DATA_BLOCK "DB242_Program8"   // DB242
{ S7_Optimized_Access := 'FALSE' }
AUTHOR : Robopac
VERSION : 0.0
// stored: AutoNumber false, IsOnlyStoredInLoadMemory false, IsWriteProtectedInAS false
   VAR RETAIN
      Program8 { S7_SetPoint := 'True'} : "DatiProgramma";
   END_VAR
BEGIN
   Program8.Wrapping := TRUE;
   Program8.TopLenght := 500;
   Program8.TopRelease := 0;
   Program8.TopDown := 0;
   Program8.Top := 4;
   Program8.PressurePTime := 0;
   Program8.LifterTime := 0;
   Program8.RevOverContrast := 1;
   Program8.RopeEndCycle := 16#02;
   Program8.Spare4 := 16#01;
   Program8.RopeTime := 1500;
   Program8.RevOverClamp := 1;
   Program8.FilmForceFinalRev := 10;
   Program8.FilmPrestretchFinalRev := 100;
   Program8.ArmSpeed := 100;
   Program8.CarriageDown4Top := 500;
   Program8.TopDownTime := 1500;
   Program8.LapsUnderTop := 0;
   Program8.Spare6 := 0;
   Program8.Spare7 := 0;
   Program8.Spare8 := 0;
   Program8.Spare9 := 0;
   Program8.Spare10 := 0;
   Program8.Spare11 := 0;
   Program8.Spare12 := 0;
   Program8.Overlap0_1 := 0;
   Program8.Height1 := 130;
   Program8.Landmark1 := FALSE;
   Program8.Lifter1 := FALSE;
   Program8.SpareBit1H1 := FALSE;
   Program8.Airblower1 := TRUE;
   Program8.NextStep1 := TRUE;
   Program8.PressureP1 := TRUE;
   Program8.SpareByte2H1 := 16#00;
   Program8.Revolution1 := 1;
   Program8.RopeUnit1_1 := 16#01;
   Program8.RopeUnit1_2 := 16#01;
   Program8.FilmForce1 := 5;
   Program8.FilmPrestretch1 := 200;
   Program8.Spare3H1 := 0;
   Program8.Spare49 := 0;
   Program8.Spare50 := 0;
   Program8.Spare51 := 0;
   Program8.Spare52 := 0;
   Program8.Spare53 := 0;
   Program8.Overlap1_2 := 0;
   Program8.Height2 := 50;
   Program8.Landmark2 := FALSE;
   Program8.Lifter2 := FALSE;
   Program8.SpareBit1H2 := FALSE;
   Program8.Airblower2 := TRUE;
   Program8.NextStep2 := TRUE;
   Program8.PressureP2 := TRUE;
   Program8.SpareByte2H2 := 16#00;
   Program8.Revolution2 := 1;
   Program8.RopeUnit2_1 := 16#01;
   Program8.RopeUnit2_2 := 16#01;
   Program8.FilmForce2 := 20;
   Program8.FilmPrestretch2 := 200;
   Program8.Spare3H2 := 0;
   Program8.Spare54 := 0;
   Program8.Spare55 := 0;
   Program8.Spare56 := 0;
   Program8.Spare57 := 0;
   Program8.Spare58 := 0;
   Program8.Overlap2_3 := 100;
   Program8.Height3 := -50;
   Program8.Landmark3 := TRUE;
   Program8.Lifter3 := FALSE;
   Program8.SpareBit1H3 := FALSE;
   Program8.Airblower3 := TRUE;
   Program8.NextStep3 := TRUE;
   Program8.PressureP3 := TRUE;
   Program8.SpareByte2H3 := 16#00;
   Program8.Revolution3 := 2;
   Program8.RopeUnit3_1 := 16#01;
   Program8.RopeUnit3_2 := 16#01;
   Program8.FilmForce3 := 30;
   Program8.FilmPrestretch3 := 200;
   Program8.Spare3H3 := 0;
   Program8.Spare59 := 0;
   Program8.Spare60 := 0;
   Program8.Spare61 := 380;
   Program8.Spare62 := 2800;
   Program8.Spare63 := 0;
   Program8.Overlap3_4 := 100;
   Program8.Height4 := 100;
   Program8.Landmark4 := FALSE;
   Program8.Lifter4 := FALSE;
   Program8.SpareBit1H4 := FALSE;
   Program8.Airblower4 := TRUE;
   Program8.NextStep4 := TRUE;
   Program8.PressureP4 := TRUE;
   Program8.SpareByte2H4 := 16#00;
   Program8.Revolution4 := 3;
   Program8.RopeUnit4_1 := 16#02;
   Program8.RopeUnit4_2 := 16#02;
   Program8.FilmForce4 := 30;
   Program8.FilmPrestretch4 := 200;
   Program8.Spare3H4 := 0;
   Program8.Spare64 := 0;
   Program8.Spare65 := 0;
   Program8.Spare66 := 0;
   Program8.Spare67 := 0;
   Program8.Spare68 := 0;
   Program8.Overlap4_5 := 0;
   Program8.Height5 := 50;
   Program8.Landmark5 := FALSE;
   Program8.Lifter5 := FALSE;
   Program8.SpareBit1H5 := FALSE;
   Program8.Airblower5 := TRUE;
   Program8.NextStep5 := FALSE;
   Program8.PressureP5 := FALSE;
   Program8.SpareByte2H5 := 16#00;
   Program8.Revolution5 := 1;
   Program8.RopeUnit5_1 := 16#01;
   Program8.RopeUnit5_2 := 16#01;
   Program8.FilmForce5 := 30;
   Program8.FilmPrestretch5 := 200;
   Program8.Spare3H5 := 0;
   Program8.Spare69 := 0;
   Program8.Spare70 := 0;
   Program8.Spare71 := 0;
   Program8.Spare72 := 0;
   Program8.Spare73 := 0;
   Program8.Overlap5_6 := 100;
   Program8.Height6 := 50;
   Program8.Landmark6 := FALSE;
   Program8.Lifter6 := FALSE;
   Program8.SpareBit1H6 := FALSE;
   Program8.Airblower6 := TRUE;
   Program8.NextStep6 := FALSE;
   Program8.PressureP6 := FALSE;
   Program8.SpareByte2H6 := 16#00;
   Program8.Revolution6 := 2;
   Program8.RopeUnit6_1 := 16#02;
   Program8.RopeUnit6_2 := 16#01;
   Program8.FilmForce6 := 20;
   Program8.FilmPrestretch6 := 200;
   Program8.Spare3H6 := 0;
   Program8.Spare74 := 0;
   Program8.Spare75 := 0;
   Program8.Spare76 := 0;
   Program8.Spare77 := 0;
   Program8.Spare78 := 0;
   Program8.Overlap6_7 := 0;
   Program8.Height7 := 0;
   Program8.Landmark7 := FALSE;
   Program8.Lifter7 := FALSE;
   Program8.SpareBit1H7 := FALSE;
   Program8.Airblower7 := FALSE;
   Program8.NextStep7 := TRUE;
   Program8.PressureP7 := FALSE;
   Program8.SpareByte2H7 := 16#00;
   Program8.Revolution7 := 1;
   Program8.RopeUnit7_1 := 16#01;
   Program8.RopeUnit7_2 := 16#01;
   Program8.FilmForce7 := 0;
   Program8.FilmPrestretch7 := 100;
   Program8.Spare3H7 := 0;
   Program8.Spare79 := 0;
   Program8.Spare80 := 0;
   Program8.Spare81 := 0;
   Program8.Spare82 := 0;
   Program8.Spare83 := 0;
   Program8.Overlap7_8 := 0;
   Program8.Height8 := 0;
   Program8.Landmark8 := FALSE;
   Program8.Lifter8 := FALSE;
   Program8.SpareBit1H8 := FALSE;
   Program8.Airblower8 := FALSE;
   Program8.NextStep8 := TRUE;
   Program8.PressureP8 := FALSE;
   Program8.SpareByte2H8 := 16#00;
   Program8.Revolution8 := 1;
   Program8.RopeUnit8_1 := 16#01;
   Program8.RopeUnit8_2 := 16#01;
   Program8.FilmForce8 := 0;
   Program8.FilmPrestretch8 := 100;
   Program8.Spare3H8 := 0;
   Program8.Spare84 := 0;
   Program8.Spare85 := 0;
   Program8.Spare86 := 0;
   Program8.Spare87 := 0;
   Program8.Spare88 := 0;
   Program8.Overlap8_9 := 0;
   Program8.Height9 := 0;
   Program8.Landmark9 := FALSE;
   Program8.Lifter9 := FALSE;
   Program8.SpareBit1H9 := FALSE;
   Program8.Airblower9 := FALSE;
   Program8.NextStep9 := TRUE;
   Program8.PressureP9 := FALSE;
   Program8.SpareByte2H9 := 16#00;
   Program8.Revolution9 := 1;
   Program8.RopeUnit9_1 := 16#01;
   Program8.RopeUnit9_2 := 16#01;
   Program8.FilmForce9 := 0;
   Program8.FilmPrestretch9 := 100;
   Program8.Spare3H9 := 0;
   Program8.Spare89 := 0;
   Program8.Spare90 := 0;
   Program8.Spare91 := 0;
   Program8.Spare92 := 0;
   Program8.Spare93 := 0;
   Program8.Overlap9_10 := 0;
   Program8.Height10 := 0;
   Program8.Landmark10 := FALSE;
   Program8.Lifter10 := FALSE;
   Program8.SpareBit1H10 := FALSE;
   Program8.Airblower10 := FALSE;
   Program8.NextStep10 := FALSE;
   Program8.PressureP10 := FALSE;
   Program8.SpareByte2H10 := 16#00;
   Program8.Revolution10 := 1;
   Program8.RopeUnit10_1 := 16#01;
   Program8.RopeUnit10_2 := 16#01;
   Program8.FilmForce10 := 0;
   Program8.FilmPrestretch10 := 100;
   Program8.Spare3H10 := 0;
   Program8.Spare94 := 0;
   Program8.Spare95 := 0;
   Program8.Spare96 := 0;
   Program8.Spare97 := 0;
   Program8.Spare98 := 0;
   Program8.Overlap10_11 := 0;
   Program8.Height11 := 0;
   Program8.Landmark11 := FALSE;
   Program8.Lifter11 := FALSE;
   Program8.SpareBit1H11 := FALSE;
   Program8.Airblower11 := FALSE;
   Program8.NextStep11 := TRUE;
   Program8.PressureP11 := FALSE;
   Program8.SpareByte2H11 := 16#00;
   Program8.Revolution11 := 1;
   Program8.RopeUnit11_1 := 16#01;
   Program8.RopeUnit11_2 := 16#01;
   Program8.FilmForce11 := 0;
   Program8.FilmPrestretch11 := 100;
   Program8.Spare3H11 := 0;
   Program8.Spare99 := 0;
   Program8.Spare100 := 0;
   Program8.Spare101 := 0;
   Program8.Spare102 := 0;
   Program8.Spare103 := 0;
   Program8.Overlap11_12 := 0;
   Program8.Height12 := 0;
   Program8.Landmark12 := FALSE;
   Program8.Lifter12 := FALSE;
   Program8.SpareBit1H12 := FALSE;
   Program8.Airblower12 := FALSE;
   Program8.NextStep12 := FALSE;
   Program8.PressureP12 := FALSE;
   Program8.SpareByte2H12 := 16#00;
   Program8.Revolution12 := 1;
   Program8.RopeUnit12_1 := 16#01;
   Program8.RopeUnit12_2 := 16#01;
   Program8.FilmForce12 := 0;
   Program8.FilmPrestretch12 := 100;
   Program8.Spare3H12 := 0;
   Program8.Spare104 := 0;
   Program8.Spare105 := 0;
   Program8.Spare106 := 0;
   Program8.Spare107 := 0;
   Program8.Spare108 := 0;
END_DATA_BLOCK

DATA_BLOCK "DB244_Program6"   // DB244
{ S7_Optimized_Access := 'FALSE' }
AUTHOR : Robopac
VERSION : 0.0
// stored: AutoNumber false, IsOnlyStoredInLoadMemory false, IsWriteProtectedInAS false
   VAR RETAIN
      Program6 { S7_SetPoint := 'True'} : "DatiProgramma";
   END_VAR
BEGIN
   Program6.Wrapping := TRUE;
   Program6.TopLenght := 500;
   Program6.TopRelease := 0;
   Program6.TopDown := 0;
   Program6.Top := 4;
   Program6.PressurePTime := 0;
   Program6.LifterTime := 0;
   Program6.RevOverContrast := 1;
   Program6.RopeEndCycle := 16#02;
   Program6.Spare4 := 16#01;
   Program6.RopeTime := 1500;
   Program6.RevOverClamp := 1;
   Program6.FilmForceFinalRev := 10;
   Program6.FilmPrestretchFinalRev := 100;
   Program6.ArmSpeed := 100;
   Program6.CarriageDown4Top := 500;
   Program6.TopDownTime := 1500;
   Program6.LapsUnderTop := 0;
   Program6.Spare6 := 0;
   Program6.Spare7 := 0;
   Program6.Spare8 := 0;
   Program6.Spare9 := 0;
   Program6.Spare10 := 0;
   Program6.Spare11 := 0;
   Program6.Spare12 := 0;
   Program6.Overlap0_1 := 0;
   Program6.Height1 := 130;
   Program6.Landmark1 := FALSE;
   Program6.Lifter1 := FALSE;
   Program6.SpareBit1H1 := FALSE;
   Program6.Airblower1 := TRUE;
   Program6.NextStep1 := TRUE;
   Program6.PressureP1 := TRUE;
   Program6.SpareByte2H1 := 16#00;
   Program6.Revolution1 := 1;
   Program6.RopeUnit1_1 := 16#01;
   Program6.RopeUnit1_2 := 16#01;
   Program6.FilmForce1 := 5;
   Program6.FilmPrestretch1 := 200;
   Program6.Spare3H1 := 0;
   Program6.Spare49 := 0;
   Program6.Spare50 := 0;
   Program6.Spare51 := 0;
   Program6.Spare52 := 0;
   Program6.Spare53 := 0;
   Program6.Overlap1_2 := 0;
   Program6.Height2 := 50;
   Program6.Landmark2 := FALSE;
   Program6.Lifter2 := FALSE;
   Program6.SpareBit1H2 := FALSE;
   Program6.Airblower2 := TRUE;
   Program6.NextStep2 := TRUE;
   Program6.PressureP2 := TRUE;
   Program6.SpareByte2H2 := 16#00;
   Program6.Revolution2 := 1;
   Program6.RopeUnit2_1 := 16#01;
   Program6.RopeUnit2_2 := 16#01;
   Program6.FilmForce2 := 20;
   Program6.FilmPrestretch2 := 200;
   Program6.Spare3H2 := 0;
   Program6.Spare54 := 0;
   Program6.Spare55 := 0;
   Program6.Spare56 := 0;
   Program6.Spare57 := 0;
   Program6.Spare58 := 0;
   Program6.Overlap2_3 := 100;
   Program6.Height3 := -50;
   Program6.Landmark3 := TRUE;
   Program6.Lifter3 := FALSE;
   Program6.SpareBit1H3 := FALSE;
   Program6.Airblower3 := TRUE;
   Program6.NextStep3 := TRUE;
   Program6.PressureP3 := TRUE;
   Program6.SpareByte2H3 := 16#00;
   Program6.Revolution3 := 2;
   Program6.RopeUnit3_1 := 16#01;
   Program6.RopeUnit3_2 := 16#01;
   Program6.FilmForce3 := 30;
   Program6.FilmPrestretch3 := 200;
   Program6.Spare3H3 := 0;
   Program6.Spare59 := 0;
   Program6.Spare60 := 0;
   Program6.Spare61 := 380;
   Program6.Spare62 := 2800;
   Program6.Spare63 := 0;
   Program6.Overlap3_4 := 100;
   Program6.Height4 := 100;
   Program6.Landmark4 := FALSE;
   Program6.Lifter4 := FALSE;
   Program6.SpareBit1H4 := FALSE;
   Program6.Airblower4 := TRUE;
   Program6.NextStep4 := TRUE;
   Program6.PressureP4 := TRUE;
   Program6.SpareByte2H4 := 16#00;
   Program6.Revolution4 := 3;
   Program6.RopeUnit4_1 := 16#02;
   Program6.RopeUnit4_2 := 16#02;
   Program6.FilmForce4 := 30;
   Program6.FilmPrestretch4 := 200;
   Program6.Spare3H4 := 0;
   Program6.Spare64 := 0;
   Program6.Spare65 := 0;
   Program6.Spare66 := 0;
   Program6.Spare67 := 0;
   Program6.Spare68 := 0;
   Program6.Overlap4_5 := 0;
   Program6.Height5 := 50;
   Program6.Landmark5 := FALSE;
   Program6.Lifter5 := FALSE;
   Program6.SpareBit1H5 := FALSE;
   Program6.Airblower5 := TRUE;
   Program6.NextStep5 := FALSE;
   Program6.PressureP5 := FALSE;
   Program6.SpareByte2H5 := 16#00;
   Program6.Revolution5 := 1;
   Program6.RopeUnit5_1 := 16#01;
   Program6.RopeUnit5_2 := 16#01;
   Program6.FilmForce5 := 30;
   Program6.FilmPrestretch5 := 200;
   Program6.Spare3H5 := 0;
   Program6.Spare69 := 0;
   Program6.Spare70 := 0;
   Program6.Spare71 := 0;
   Program6.Spare72 := 0;
   Program6.Spare73 := 0;
   Program6.Overlap5_6 := 100;
   Program6.Height6 := 50;
   Program6.Landmark6 := FALSE;
   Program6.Lifter6 := FALSE;
   Program6.SpareBit1H6 := FALSE;
   Program6.Airblower6 := TRUE;
   Program6.NextStep6 := FALSE;
   Program6.PressureP6 := FALSE;
   Program6.SpareByte2H6 := 16#00;
   Program6.Revolution6 := 2;
   Program6.RopeUnit6_1 := 16#02;
   Program6.RopeUnit6_2 := 16#01;
   Program6.FilmForce6 := 20;
   Program6.FilmPrestretch6 := 200;
   Program6.Spare3H6 := 0;
   Program6.Spare74 := 0;
   Program6.Spare75 := 0;
   Program6.Spare76 := 0;
   Program6.Spare77 := 0;
   Program6.Spare78 := 0;
   Program6.Overlap6_7 := 0;
   Program6.Height7 := 0;
   Program6.Landmark7 := FALSE;
   Program6.Lifter7 := FALSE;
   Program6.SpareBit1H7 := FALSE;
   Program6.Airblower7 := FALSE;
   Program6.NextStep7 := TRUE;
   Program6.PressureP7 := FALSE;
   Program6.SpareByte2H7 := 16#00;
   Program6.Revolution7 := 1;
   Program6.RopeUnit7_1 := 16#01;
   Program6.RopeUnit7_2 := 16#01;
   Program6.FilmForce7 := 0;
   Program6.FilmPrestretch7 := 100;
   Program6.Spare3H7 := 0;
   Program6.Spare79 := 0;
   Program6.Spare80 := 0;
   Program6.Spare81 := 0;
   Program6.Spare82 := 0;
   Program6.Spare83 := 0;
   Program6.Overlap7_8 := 0;
   Program6.Height8 := 0;
   Program6.Landmark8 := FALSE;
   Program6.Lifter8 := FALSE;
   Program6.SpareBit1H8 := FALSE;
   Program6.Airblower8 := FALSE;
   Program6.NextStep8 := TRUE;
   Program6.PressureP8 := FALSE;
   Program6.SpareByte2H8 := 16#00;
   Program6.Revolution8 := 1;
   Program6.RopeUnit8_1 := 16#01;
   Program6.RopeUnit8_2 := 16#01;
   Program6.FilmForce8 := 0;
   Program6.FilmPrestretch8 := 100;
   Program6.Spare3H8 := 0;
   Program6.Spare84 := 0;
   Program6.Spare85 := 0;
   Program6.Spare86 := 0;
   Program6.Spare87 := 0;
   Program6.Spare88 := 0;
   Program6.Overlap8_9 := 0;
   Program6.Height9 := 0;
   Program6.Landmark9 := FALSE;
   Program6.Lifter9 := FALSE;
   Program6.SpareBit1H9 := FALSE;
   Program6.Airblower9 := FALSE;
   Program6.NextStep9 := TRUE;
   Program6.PressureP9 := FALSE;
   Program6.SpareByte2H9 := 16#00;
   Program6.Revolution9 := 1;
   Program6.RopeUnit9_1 := 16#01;
   Program6.RopeUnit9_2 := 16#01;
   Program6.FilmForce9 := 0;
   Program6.FilmPrestretch9 := 100;
   Program6.Spare3H9 := 0;
   Program6.Spare89 := 0;
   Program6.Spare90 := 0;
   Program6.Spare91 := 0;
   Program6.Spare92 := 0;
   Program6.Spare93 := 0;
   Program6.Overlap9_10 := 0;
   Program6.Height10 := 0;
   Program6.Landmark10 := FALSE;
   Program6.Lifter10 := FALSE;
   Program6.SpareBit1H10 := FALSE;
   Program6.Airblower10 := FALSE;
   Program6.NextStep10 := FALSE;
   Program6.PressureP10 := FALSE;
   Program6.SpareByte2H10 := 16#00;
   Program6.Revolution10 := 1;
   Program6.RopeUnit10_1 := 16#01;
   Program6.RopeUnit10_2 := 16#01;
   Program6.FilmForce10 := 0;
   Program6.FilmPrestretch10 := 100;
   Program6.Spare3H10 := 0;
   Program6.Spare94 := 0;
   Program6.Spare95 := 0;
   Program6.Spare96 := 0;
   Program6.Spare97 := 0;
   Program6.Spare98 := 0;
   Program6.Overlap10_11 := 0;
   Program6.Height11 := 0;
   Program6.Landmark11 := FALSE;
   Program6.Lifter11 := FALSE;
   Program6.SpareBit1H11 := FALSE;
   Program6.Airblower11 := FALSE;
   Program6.NextStep11 := TRUE;
   Program6.PressureP11 := FALSE;
   Program6.SpareByte2H11 := 16#00;
   Program6.Revolution11 := 1;
   Program6.RopeUnit11_1 := 16#01;
   Program6.RopeUnit11_2 := 16#01;
   Program6.FilmForce11 := 0;
   Program6.FilmPrestretch11 := 100;
   Program6.Spare3H11 := 0;
   Program6.Spare99 := 0;
   Program6.Spare100 := 0;
   Program6.Spare101 := 0;
   Program6.Spare102 := 0;
   Program6.Spare103 := 0;
   Program6.Overlap11_12 := 0;
   Program6.Height12 := 0;
   Program6.Landmark12 := FALSE;
   Program6.Lifter12 := FALSE;
   Program6.SpareBit1H12 := FALSE;
   Program6.Airblower12 := FALSE;
   Program6.NextStep12 := FALSE;
   Program6.PressureP12 := FALSE;
   Program6.SpareByte2H12 := 16#00;
   Program6.Revolution12 := 1;
   Program6.RopeUnit12_1 := 16#01;
   Program6.RopeUnit12_2 := 16#01;
   Program6.FilmForce12 := 0;
   Program6.FilmPrestretch12 := 100;
   Program6.Spare3H12 := 0;
   Program6.Spare104 := 0;
   Program6.Spare105 := 0;
   Program6.Spare106 := 0;
   Program6.Spare107 := 0;
   Program6.Spare108 := 0;
END_DATA_BLOCK

DATA_BLOCK "DB245_Program5"   // DB245
{ S7_Optimized_Access := 'FALSE' }
AUTHOR : Robopac
VERSION : 0.0
// stored: AutoNumber false, IsOnlyStoredInLoadMemory false, IsWriteProtectedInAS false
   VAR RETAIN
      Program5 { S7_SetPoint := 'True'} : "DatiProgramma";
   END_VAR
BEGIN
   Program5.Wrapping := TRUE;
   Program5.TopLenght := 500;
   Program5.TopRelease := 0;
   Program5.TopDown := 0;
   Program5.Top := 4;
   Program5.PressurePTime := 0;
   Program5.LifterTime := 0;
   Program5.RevOverContrast := 1;
   Program5.RopeEndCycle := 16#02;
   Program5.Spare4 := 16#01;
   Program5.RopeTime := 1500;
   Program5.RevOverClamp := 1;
   Program5.FilmForceFinalRev := 10;
   Program5.FilmPrestretchFinalRev := 100;
   Program5.ArmSpeed := 100;
   Program5.CarriageDown4Top := 500;
   Program5.TopDownTime := 1500;
   Program5.LapsUnderTop := 0;
   Program5.Spare6 := 0;
   Program5.Spare7 := 0;
   Program5.Spare8 := 0;
   Program5.Spare9 := 0;
   Program5.Spare10 := 0;
   Program5.Spare11 := 0;
   Program5.Spare12 := 0;
   Program5.Overlap0_1 := 0;
   Program5.Height1 := 130;
   Program5.Landmark1 := FALSE;
   Program5.Lifter1 := FALSE;
   Program5.SpareBit1H1 := FALSE;
   Program5.Airblower1 := TRUE;
   Program5.NextStep1 := TRUE;
   Program5.PressureP1 := TRUE;
   Program5.SpareByte2H1 := 16#00;
   Program5.Revolution1 := 1;
   Program5.RopeUnit1_1 := 16#01;
   Program5.RopeUnit1_2 := 16#01;
   Program5.FilmForce1 := 5;
   Program5.FilmPrestretch1 := 200;
   Program5.Spare3H1 := 0;
   Program5.Spare49 := 0;
   Program5.Spare50 := 0;
   Program5.Spare51 := 0;
   Program5.Spare52 := 0;
   Program5.Spare53 := 0;
   Program5.Overlap1_2 := 0;
   Program5.Height2 := 50;
   Program5.Landmark2 := FALSE;
   Program5.Lifter2 := FALSE;
   Program5.SpareBit1H2 := FALSE;
   Program5.Airblower2 := TRUE;
   Program5.NextStep2 := TRUE;
   Program5.PressureP2 := TRUE;
   Program5.SpareByte2H2 := 16#00;
   Program5.Revolution2 := 1;
   Program5.RopeUnit2_1 := 16#01;
   Program5.RopeUnit2_2 := 16#01;
   Program5.FilmForce2 := 20;
   Program5.FilmPrestretch2 := 200;
   Program5.Spare3H2 := 0;
   Program5.Spare54 := 0;
   Program5.Spare55 := 0;
   Program5.Spare56 := 0;
   Program5.Spare57 := 0;
   Program5.Spare58 := 0;
   Program5.Overlap2_3 := 100;
   Program5.Height3 := -50;
   Program5.Landmark3 := TRUE;
   Program5.Lifter3 := FALSE;
   Program5.SpareBit1H3 := FALSE;
   Program5.Airblower3 := TRUE;
   Program5.NextStep3 := TRUE;
   Program5.PressureP3 := TRUE;
   Program5.SpareByte2H3 := 16#00;
   Program5.Revolution3 := 2;
   Program5.RopeUnit3_1 := 16#01;
   Program5.RopeUnit3_2 := 16#01;
   Program5.FilmForce3 := 30;
   Program5.FilmPrestretch3 := 200;
   Program5.Spare3H3 := 0;
   Program5.Spare59 := 0;
   Program5.Spare60 := 0;
   Program5.Spare61 := 380;
   Program5.Spare62 := 2800;
   Program5.Spare63 := 0;
   Program5.Overlap3_4 := 100;
   Program5.Height4 := 100;
   Program5.Landmark4 := FALSE;
   Program5.Lifter4 := FALSE;
   Program5.SpareBit1H4 := FALSE;
   Program5.Airblower4 := TRUE;
   Program5.NextStep4 := TRUE;
   Program5.PressureP4 := TRUE;
   Program5.SpareByte2H4 := 16#00;
   Program5.Revolution4 := 3;
   Program5.RopeUnit4_1 := 16#02;
   Program5.RopeUnit4_2 := 16#02;
   Program5.FilmForce4 := 30;
   Program5.FilmPrestretch4 := 200;
   Program5.Spare3H4 := 0;
   Program5.Spare64 := 0;
   Program5.Spare65 := 0;
   Program5.Spare66 := 0;
   Program5.Spare67 := 0;
   Program5.Spare68 := 0;
   Program5.Overlap4_5 := 0;
   Program5.Height5 := 50;
   Program5.Landmark5 := FALSE;
   Program5.Lifter5 := FALSE;
   Program5.SpareBit1H5 := FALSE;
   Program5.Airblower5 := TRUE;
   Program5.NextStep5 := FALSE;
   Program5.PressureP5 := FALSE;
   Program5.SpareByte2H5 := 16#00;
   Program5.Revolution5 := 1;
   Program5.RopeUnit5_1 := 16#01;
   Program5.RopeUnit5_2 := 16#01;
   Program5.FilmForce5 := 30;
   Program5.FilmPrestretch5 := 200;
   Program5.Spare3H5 := 0;
   Program5.Spare69 := 0;
   Program5.Spare70 := 0;
   Program5.Spare71 := 0;
   Program5.Spare72 := 0;
   Program5.Spare73 := 0;
   Program5.Overlap5_6 := 100;
   Program5.Height6 := 50;
   Program5.Landmark6 := FALSE;
   Program5.Lifter6 := FALSE;
   Program5.SpareBit1H6 := FALSE;
   Program5.Airblower6 := TRUE;
   Program5.NextStep6 := FALSE;
   Program5.PressureP6 := FALSE;
   Program5.SpareByte2H6 := 16#00;
   Program5.Revolution6 := 2;
   Program5.RopeUnit6_1 := 16#02;
   Program5.RopeUnit6_2 := 16#01;
   Program5.FilmForce6 := 20;
   Program5.FilmPrestretch6 := 200;
   Program5.Spare3H6 := 0;
   Program5.Spare74 := 0;
   Program5.Spare75 := 0;
   Program5.Spare76 := 0;
   Program5.Spare77 := 0;
   Program5.Spare78 := 0;
   Program5.Overlap6_7 := 0;
   Program5.Height7 := 0;
   Program5.Landmark7 := FALSE;
   Program5.Lifter7 := FALSE;
   Program5.SpareBit1H7 := FALSE;
   Program5.Airblower7 := FALSE;
   Program5.NextStep7 := TRUE;
   Program5.PressureP7 := FALSE;
   Program5.SpareByte2H7 := 16#00;
   Program5.Revolution7 := 1;
   Program5.RopeUnit7_1 := 16#01;
   Program5.RopeUnit7_2 := 16#01;
   Program5.FilmForce7 := 0;
   Program5.FilmPrestretch7 := 100;
   Program5.Spare3H7 := 0;
   Program5.Spare79 := 0;
   Program5.Spare80 := 0;
   Program5.Spare81 := 0;
   Program5.Spare82 := 0;
   Program5.Spare83 := 0;
   Program5.Overlap7_8 := 0;
   Program5.Height8 := 0;
   Program5.Landmark8 := FALSE;
   Program5.Lifter8 := FALSE;
   Program5.SpareBit1H8 := FALSE;
   Program5.Airblower8 := FALSE;
   Program5.NextStep8 := TRUE;
   Program5.PressureP8 := FALSE;
   Program5.SpareByte2H8 := 16#00;
   Program5.Revolution8 := 1;
   Program5.RopeUnit8_1 := 16#01;
   Program5.RopeUnit8_2 := 16#01;
   Program5.FilmForce8 := 0;
   Program5.FilmPrestretch8 := 100;
   Program5.Spare3H8 := 0;
   Program5.Spare84 := 0;
   Program5.Spare85 := 0;
   Program5.Spare86 := 0;
   Program5.Spare87 := 0;
   Program5.Spare88 := 0;
   Program5.Overlap8_9 := 0;
   Program5.Height9 := 0;
   Program5.Landmark9 := FALSE;
   Program5.Lifter9 := FALSE;
   Program5.SpareBit1H9 := FALSE;
   Program5.Airblower9 := FALSE;
   Program5.NextStep9 := TRUE;
   Program5.PressureP9 := FALSE;
   Program5.SpareByte2H9 := 16#00;
   Program5.Revolution9 := 1;
   Program5.RopeUnit9_1 := 16#01;
   Program5.RopeUnit9_2 := 16#01;
   Program5.FilmForce9 := 0;
   Program5.FilmPrestretch9 := 100;
   Program5.Spare3H9 := 0;
   Program5.Spare89 := 0;
   Program5.Spare90 := 0;
   Program5.Spare91 := 0;
   Program5.Spare92 := 0;
   Program5.Spare93 := 0;
   Program5.Overlap9_10 := 0;
   Program5.Height10 := 0;
   Program5.Landmark10 := FALSE;
   Program5.Lifter10 := FALSE;
   Program5.SpareBit1H10 := FALSE;
   Program5.Airblower10 := FALSE;
   Program5.NextStep10 := FALSE;
   Program5.PressureP10 := FALSE;
   Program5.SpareByte2H10 := 16#00;
   Program5.Revolution10 := 1;
   Program5.RopeUnit10_1 := 16#01;
   Program5.RopeUnit10_2 := 16#01;
   Program5.FilmForce10 := 0;
   Program5.FilmPrestretch10 := 100;
   Program5.Spare3H10 := 0;
   Program5.Spare94 := 0;
   Program5.Spare95 := 0;
   Program5.Spare96 := 0;
   Program5.Spare97 := 0;
   Program5.Spare98 := 0;
   Program5.Overlap10_11 := 0;
   Program5.Height11 := 0;
   Program5.Landmark11 := FALSE;
   Program5.Lifter11 := FALSE;
   Program5.SpareBit1H11 := FALSE;
   Program5.Airblower11 := FALSE;
   Program5.NextStep11 := TRUE;
   Program5.PressureP11 := FALSE;
   Program5.SpareByte2H11 := 16#00;
   Program5.Revolution11 := 1;
   Program5.RopeUnit11_1 := 16#01;
   Program5.RopeUnit11_2 := 16#01;
   Program5.FilmForce11 := 0;
   Program5.FilmPrestretch11 := 100;
   Program5.Spare3H11 := 0;
   Program5.Spare99 := 0;
   Program5.Spare100 := 0;
   Program5.Spare101 := 0;
   Program5.Spare102 := 0;
   Program5.Spare103 := 0;
   Program5.Overlap11_12 := 0;
   Program5.Height12 := 0;
   Program5.Landmark12 := FALSE;
   Program5.Lifter12 := FALSE;
   Program5.SpareBit1H12 := FALSE;
   Program5.Airblower12 := FALSE;
   Program5.NextStep12 := FALSE;
   Program5.PressureP12 := FALSE;
   Program5.SpareByte2H12 := 16#00;
   Program5.Revolution12 := 1;
   Program5.RopeUnit12_1 := 16#01;
   Program5.RopeUnit12_2 := 16#01;
   Program5.FilmForce12 := 0;
   Program5.FilmPrestretch12 := 100;
   Program5.Spare3H12 := 0;
   Program5.Spare104 := 0;
   Program5.Spare105 := 0;
   Program5.Spare106 := 0;
   Program5.Spare107 := 0;
   Program5.Spare108 := 0;
END_DATA_BLOCK

DATA_BLOCK "DB247_Program3"   // DB247
{ S7_Optimized_Access := 'FALSE' }
AUTHOR : Robopac
VERSION : 0.0
// stored: AutoNumber false, IsOnlyStoredInLoadMemory false, IsWriteProtectedInAS false
   VAR RETAIN
      Program3 { S7_SetPoint := 'True'} : "DatiProgramma";
   END_VAR
BEGIN
   Program3.Wrapping := TRUE;
   Program3.TopLenght := 500;
   Program3.TopRelease := 0;
   Program3.TopDown := 0;
   Program3.Top := 4;
   Program3.PressurePTime := 0;
   Program3.LifterTime := 0;
   Program3.RevOverContrast := 1;
   Program3.RopeEndCycle := 16#01;
   Program3.Spare4 := 16#01;
   Program3.RopeTime := 1500;
   Program3.RevOverClamp := 1;
   Program3.FilmForceFinalRev := 20;
   Program3.FilmPrestretchFinalRev := 100;
   Program3.ArmSpeed := 90;
   Program3.CarriageDown4Top := 500;
   Program3.TopDownTime := 1500;
   Program3.LapsUnderTop := 0;
   Program3.Spare6 := 0;
   Program3.Spare7 := 0;
   Program3.Spare8 := 0;
   Program3.Spare9 := 0;
   Program3.Spare10 := 0;
   Program3.Spare11 := 0;
   Program3.Spare12 := 0;
   Program3.Overlap0_1 := 0;
   Program3.Height1 := 120;
   Program3.Landmark1 := FALSE;
   Program3.Lifter1 := FALSE;
   Program3.SpareBit1H1 := FALSE;
   Program3.Airblower1 := TRUE;
   Program3.NextStep1 := TRUE;
   Program3.PressureP1 := TRUE;
   Program3.SpareByte2H1 := 16#00;
   Program3.Revolution1 := 1;
   Program3.RopeUnit1_1 := 16#01;
   Program3.RopeUnit1_2 := 16#01;
   Program3.FilmForce1 := 5;
   Program3.FilmPrestretch1 := 200;
   Program3.Spare3H1 := 0;
   Program3.Spare49 := 0;
   Program3.Spare50 := 0;
   Program3.Spare51 := 0;
   Program3.Spare52 := 0;
   Program3.Spare53 := 0;
   Program3.Overlap1_2 := 0;
   Program3.Height2 := 60;
   Program3.Landmark2 := FALSE;
   Program3.Lifter2 := FALSE;
   Program3.SpareBit1H2 := FALSE;
   Program3.Airblower2 := TRUE;
   Program3.NextStep2 := TRUE;
   Program3.PressureP2 := TRUE;
   Program3.SpareByte2H2 := 16#00;
   Program3.Revolution2 := 3;
   Program3.RopeUnit2_1 := 16#01;
   Program3.RopeUnit2_2 := 16#01;
   Program3.FilmForce2 := 10;
   Program3.FilmPrestretch2 := 200;
   Program3.Spare3H2 := 0;
   Program3.Spare54 := 0;
   Program3.Spare55 := 0;
   Program3.Spare56 := 0;
   Program3.Spare57 := 0;
   Program3.Spare58 := 0;
   Program3.Overlap2_3 := 100;
   Program3.Height3 := 120;
   Program3.Landmark3 := FALSE;
   Program3.Lifter3 := FALSE;
   Program3.SpareBit1H3 := FALSE;
   Program3.Airblower3 := TRUE;
   Program3.NextStep3 := TRUE;
   Program3.PressureP3 := TRUE;
   Program3.SpareByte2H3 := 16#00;
   Program3.Revolution3 := 2;
   Program3.RopeUnit3_1 := 16#01;
   Program3.RopeUnit3_2 := 16#01;
   Program3.FilmForce3 := 5;
   Program3.FilmPrestretch3 := 200;
   Program3.Spare3H3 := 0;
   Program3.Spare59 := 0;
   Program3.Spare60 := 0;
   Program3.Spare61 := 380;
   Program3.Spare62 := 2800;
   Program3.Spare63 := 0;
   Program3.Overlap3_4 := 200;
   Program3.Height4 := 120;
   Program3.Landmark4 := FALSE;
   Program3.Lifter4 := FALSE;
   Program3.SpareBit1H4 := FALSE;
   Program3.Airblower4 := TRUE;
   Program3.NextStep4 := TRUE;
   Program3.PressureP4 := TRUE;
   Program3.SpareByte2H4 := 16#00;
   Program3.Revolution4 := 1;
   Program3.RopeUnit4_1 := 16#01;
   Program3.RopeUnit4_2 := 16#01;
   Program3.FilmForce4 := 20;
   Program3.FilmPrestretch4 := 200;
   Program3.Spare3H4 := 0;
   Program3.Spare64 := 0;
   Program3.Spare65 := 0;
   Program3.Spare66 := 0;
   Program3.Spare67 := 0;
   Program3.Spare68 := 0;
   Program3.Overlap4_5 := 200;
   Program3.Height5 := -150;
   Program3.Landmark5 := TRUE;
   Program3.Lifter5 := FALSE;
   Program3.SpareBit1H5 := FALSE;
   Program3.Airblower5 := FALSE;
   Program3.NextStep5 := TRUE;
   Program3.PressureP5 := FALSE;
   Program3.SpareByte2H5 := 16#00;
   Program3.Revolution5 := 1;
   Program3.RopeUnit5_1 := 16#01;
   Program3.RopeUnit5_2 := 16#01;
   Program3.FilmForce5 := 20;
   Program3.FilmPrestretch5 := 200;
   Program3.Spare3H5 := 0;
   Program3.Spare69 := 0;
   Program3.Spare70 := 0;
   Program3.Spare71 := 0;
   Program3.Spare72 := 0;
   Program3.Spare73 := 0;
   Program3.Overlap5_6 := 100;
   Program3.Height6 := 0;
   Program3.Landmark6 := FALSE;
   Program3.Lifter6 := FALSE;
   Program3.SpareBit1H6 := FALSE;
   Program3.Airblower6 := FALSE;
   Program3.NextStep6 := FALSE;
   Program3.PressureP6 := FALSE;
   Program3.SpareByte2H6 := 16#00;
   Program3.Revolution6 := 1;
   Program3.RopeUnit6_1 := 16#01;
   Program3.RopeUnit6_2 := 16#01;
   Program3.FilmForce6 := 30;
   Program3.FilmPrestretch6 := 200;
   Program3.Spare3H6 := 0;
   Program3.Spare74 := 0;
   Program3.Spare75 := 0;
   Program3.Spare76 := 0;
   Program3.Spare77 := 0;
   Program3.Spare78 := 0;
   Program3.Overlap6_7 := 0;
   Program3.Height7 := 0;
   Program3.Landmark7 := FALSE;
   Program3.Lifter7 := FALSE;
   Program3.SpareBit1H7 := FALSE;
   Program3.Airblower7 := FALSE;
   Program3.NextStep7 := TRUE;
   Program3.PressureP7 := FALSE;
   Program3.SpareByte2H7 := 16#00;
   Program3.Revolution7 := 1;
   Program3.RopeUnit7_1 := 16#01;
   Program3.RopeUnit7_2 := 16#01;
   Program3.FilmForce7 := 0;
   Program3.FilmPrestretch7 := 100;
   Program3.Spare3H7 := 0;
   Program3.Spare79 := 0;
   Program3.Spare80 := 0;
   Program3.Spare81 := 0;
   Program3.Spare82 := 0;
   Program3.Spare83 := 0;
   Program3.Overlap7_8 := 0;
   Program3.Height8 := 0;
   Program3.Landmark8 := FALSE;
   Program3.Lifter8 := FALSE;
   Program3.SpareBit1H8 := FALSE;
   Program3.Airblower8 := FALSE;
   Program3.NextStep8 := TRUE;
   Program3.PressureP8 := FALSE;
   Program3.SpareByte2H8 := 16#00;
   Program3.Revolution8 := 1;
   Program3.RopeUnit8_1 := 16#01;
   Program3.RopeUnit8_2 := 16#01;
   Program3.FilmForce8 := 0;
   Program3.FilmPrestretch8 := 100;
   Program3.Spare3H8 := 0;
   Program3.Spare84 := 0;
   Program3.Spare85 := 0;
   Program3.Spare86 := 0;
   Program3.Spare87 := 0;
   Program3.Spare88 := 0;
   Program3.Overlap8_9 := 0;
   Program3.Height9 := 0;
   Program3.Landmark9 := FALSE;
   Program3.Lifter9 := FALSE;
   Program3.SpareBit1H9 := FALSE;
   Program3.Airblower9 := FALSE;
   Program3.NextStep9 := TRUE;
   Program3.PressureP9 := FALSE;
   Program3.SpareByte2H9 := 16#00;
   Program3.Revolution9 := 1;
   Program3.RopeUnit9_1 := 16#01;
   Program3.RopeUnit9_2 := 16#01;
   Program3.FilmForce9 := 0;
   Program3.FilmPrestretch9 := 100;
   Program3.Spare3H9 := 0;
   Program3.Spare89 := 0;
   Program3.Spare90 := 0;
   Program3.Spare91 := 0;
   Program3.Spare92 := 0;
   Program3.Spare93 := 0;
   Program3.Overlap9_10 := 0;
   Program3.Height10 := 0;
   Program3.Landmark10 := FALSE;
   Program3.Lifter10 := FALSE;
   Program3.SpareBit1H10 := FALSE;
   Program3.Airblower10 := FALSE;
   Program3.NextStep10 := FALSE;
   Program3.PressureP10 := FALSE;
   Program3.SpareByte2H10 := 16#00;
   Program3.Revolution10 := 1;
   Program3.RopeUnit10_1 := 16#01;
   Program3.RopeUnit10_2 := 16#01;
   Program3.FilmForce10 := 0;
   Program3.FilmPrestretch10 := 100;
   Program3.Spare3H10 := 0;
   Program3.Spare94 := 0;
   Program3.Spare95 := 0;
   Program3.Spare96 := 0;
   Program3.Spare97 := 0;
   Program3.Spare98 := 0;
   Program3.Overlap10_11 := 0;
   Program3.Height11 := 0;
   Program3.Landmark11 := FALSE;
   Program3.Lifter11 := FALSE;
   Program3.SpareBit1H11 := FALSE;
   Program3.Airblower11 := FALSE;
   Program3.NextStep11 := TRUE;
   Program3.PressureP11 := FALSE;
   Program3.SpareByte2H11 := 16#00;
   Program3.Revolution11 := 1;
   Program3.RopeUnit11_1 := 16#01;
   Program3.RopeUnit11_2 := 16#01;
   Program3.FilmForce11 := 0;
   Program3.FilmPrestretch11 := 100;
   Program3.Spare3H11 := 0;
   Program3.Spare99 := 0;
   Program3.Spare100 := 0;
   Program3.Spare101 := 0;
   Program3.Spare102 := 0;
   Program3.Spare103 := 0;
   Program3.Overlap11_12 := 0;
   Program3.Height12 := 0;
   Program3.Landmark12 := FALSE;
   Program3.Lifter12 := FALSE;
   Program3.SpareBit1H12 := FALSE;
   Program3.Airblower12 := FALSE;
   Program3.NextStep12 := FALSE;
   Program3.PressureP12 := FALSE;
   Program3.SpareByte2H12 := 16#00;
   Program3.Revolution12 := 1;
   Program3.RopeUnit12_1 := 16#01;
   Program3.RopeUnit12_2 := 16#01;
   Program3.FilmForce12 := 0;
   Program3.FilmPrestretch12 := 100;
   Program3.Spare3H12 := 0;
   Program3.Spare104 := 0;
   Program3.Spare105 := 0;
   Program3.Spare106 := 0;
   Program3.Spare107 := 0;
   Program3.Spare108 := 0;
END_DATA_BLOCK

DATA_BLOCK "DB248_Program2"   // DB248
{ S7_Optimized_Access := 'FALSE' }
AUTHOR : Robopac
VERSION : 0.0
// stored: AutoNumber false, IsOnlyStoredInLoadMemory false, IsWriteProtectedInAS false
   VAR RETAIN
      Program2 { S7_SetPoint := 'True'} : "DatiProgramma";
   END_VAR
BEGIN
   Program2.Wrapping := TRUE;
   Program2.TopLenght := 500;
   Program2.TopRelease := 0;
   Program2.TopDown := 0;
   Program2.Top := 4;
   Program2.PressurePTime := 0;
   Program2.LifterTime := 0;
   Program2.RevOverContrast := 1;
   Program2.RopeEndCycle := 16#01;
   Program2.Spare4 := 16#01;
   Program2.RopeTime := 1500;
   Program2.RevOverClamp := 1;
   Program2.FilmForceFinalRev := 35;
   Program2.FilmPrestretchFinalRev := 100;
   Program2.ArmSpeed := 85;
   Program2.CarriageDown4Top := 500;
   Program2.TopDownTime := 1500;
   Program2.LapsUnderTop := 0;
   Program2.Spare6 := 0;
   Program2.Spare7 := 0;
   Program2.Spare8 := 0;
   Program2.Spare9 := 0;
   Program2.Spare10 := 0;
   Program2.Spare11 := 0;
   Program2.Spare12 := 0;
   Program2.Overlap0_1 := 0;
   Program2.Height1 := 180;
   Program2.Landmark1 := FALSE;
   Program2.Lifter1 := FALSE;
   Program2.SpareBit1H1 := FALSE;
   Program2.Airblower1 := TRUE;
   Program2.NextStep1 := TRUE;
   Program2.PressureP1 := TRUE;
   Program2.SpareByte2H1 := 16#00;
   Program2.Revolution1 := 1;
   Program2.RopeUnit1_1 := 16#01;
   Program2.RopeUnit1_2 := 16#01;
   Program2.FilmForce1 := 5;
   Program2.FilmPrestretch1 := 200;
   Program2.Spare3H1 := 0;
   Program2.Spare49 := 0;
   Program2.Spare50 := 0;
   Program2.Spare51 := 0;
   Program2.Spare52 := 0;
   Program2.Spare53 := 0;
   Program2.Overlap1_2 := 200;
   Program2.Height2 := -100;
   Program2.Landmark2 := TRUE;
   Program2.Lifter2 := FALSE;
   Program2.SpareBit1H2 := FALSE;
   Program2.Airblower2 := TRUE;
   Program2.NextStep2 := TRUE;
   Program2.PressureP2 := TRUE;
   Program2.SpareByte2H2 := 16#00;
   Program2.Revolution2 := 2;
   Program2.RopeUnit2_1 := 16#01;
   Program2.RopeUnit2_2 := 16#01;
   Program2.FilmForce2 := 20;
   Program2.FilmPrestretch2 := 200;
   Program2.Spare3H2 := 0;
   Program2.Spare54 := 0;
   Program2.Spare55 := 0;
   Program2.Spare56 := 0;
   Program2.Spare57 := 0;
   Program2.Spare58 := 0;
   Program2.Overlap2_3 := 200;
   Program2.Height3 := 80;
   Program2.Landmark3 := FALSE;
   Program2.Lifter3 := FALSE;
   Program2.SpareBit1H3 := FALSE;
   Program2.Airblower3 := TRUE;
   Program2.NextStep3 := TRUE;
   Program2.PressureP3 := TRUE;
   Program2.SpareByte2H3 := 16#00;
   Program2.Revolution3 := 2;
   Program2.RopeUnit3_1 := 16#01;
   Program2.RopeUnit3_2 := 16#01;
   Program2.FilmForce3 := 10;
   Program2.FilmPrestretch3 := 200;
   Program2.Spare3H3 := 0;
   Program2.Spare59 := 0;
   Program2.Spare60 := 0;
   Program2.Spare61 := 380;
   Program2.Spare62 := 2800;
   Program2.Spare63 := 0;
   Program2.Overlap3_4 := 200;
   Program2.Height4 := 120;
   Program2.Landmark4 := FALSE;
   Program2.Lifter4 := FALSE;
   Program2.SpareBit1H4 := FALSE;
   Program2.Airblower4 := TRUE;
   Program2.NextStep4 := TRUE;
   Program2.PressureP4 := TRUE;
   Program2.SpareByte2H4 := 16#00;
   Program2.Revolution4 := 2;
   Program2.RopeUnit4_1 := 16#02;
   Program2.RopeUnit4_2 := 16#02;
   Program2.FilmForce4 := 20;
   Program2.FilmPrestretch4 := 200;
   Program2.Spare3H4 := 0;
   Program2.Spare64 := 0;
   Program2.Spare65 := 0;
   Program2.Spare66 := 0;
   Program2.Spare67 := 0;
   Program2.Spare68 := 0;
   Program2.Overlap4_5 := 200;
   Program2.Height5 := 90;
   Program2.Landmark5 := FALSE;
   Program2.Lifter5 := FALSE;
   Program2.SpareBit1H5 := FALSE;
   Program2.Airblower5 := TRUE;
   Program2.NextStep5 := FALSE;
   Program2.PressureP5 := FALSE;
   Program2.SpareByte2H5 := 16#00;
   Program2.Revolution5 := 1;
   Program2.RopeUnit5_1 := 16#01;
   Program2.RopeUnit5_2 := 16#01;
   Program2.FilmForce5 := 20;
   Program2.FilmPrestretch5 := 200;
   Program2.Spare3H5 := 0;
   Program2.Spare69 := 0;
   Program2.Spare70 := 0;
   Program2.Spare71 := 0;
   Program2.Spare72 := 0;
   Program2.Spare73 := 0;
   Program2.Overlap5_6 := 300;
   Program2.Height6 := 120;
   Program2.Landmark6 := FALSE;
   Program2.Lifter6 := FALSE;
   Program2.SpareBit1H6 := FALSE;
   Program2.Airblower6 := TRUE;
   Program2.NextStep6 := FALSE;
   Program2.PressureP6 := FALSE;
   Program2.SpareByte2H6 := 16#00;
   Program2.Revolution6 := 1;
   Program2.RopeUnit6_1 := 16#01;
   Program2.RopeUnit6_2 := 16#01;
   Program2.FilmForce6 := 20;
   Program2.FilmPrestretch6 := 200;
   Program2.Spare3H6 := 0;
   Program2.Spare74 := 0;
   Program2.Spare75 := 0;
   Program2.Spare76 := 0;
   Program2.Spare77 := 0;
   Program2.Spare78 := 0;
   Program2.Overlap6_7 := 0;
   Program2.Height7 := 0;
   Program2.Landmark7 := FALSE;
   Program2.Lifter7 := FALSE;
   Program2.SpareBit1H7 := FALSE;
   Program2.Airblower7 := FALSE;
   Program2.NextStep7 := TRUE;
   Program2.PressureP7 := FALSE;
   Program2.SpareByte2H7 := 16#00;
   Program2.Revolution7 := 1;
   Program2.RopeUnit7_1 := 16#01;
   Program2.RopeUnit7_2 := 16#01;
   Program2.FilmForce7 := 0;
   Program2.FilmPrestretch7 := 100;
   Program2.Spare3H7 := 0;
   Program2.Spare79 := 0;
   Program2.Spare80 := 0;
   Program2.Spare81 := 0;
   Program2.Spare82 := 0;
   Program2.Spare83 := 0;
   Program2.Overlap7_8 := 0;
   Program2.Height8 := 0;
   Program2.Landmark8 := FALSE;
   Program2.Lifter8 := FALSE;
   Program2.SpareBit1H8 := FALSE;
   Program2.Airblower8 := FALSE;
   Program2.NextStep8 := TRUE;
   Program2.PressureP8 := FALSE;
   Program2.SpareByte2H8 := 16#00;
   Program2.Revolution8 := 1;
   Program2.RopeUnit8_1 := 16#01;
   Program2.RopeUnit8_2 := 16#01;
   Program2.FilmForce8 := 0;
   Program2.FilmPrestretch8 := 100;
   Program2.Spare3H8 := 0;
   Program2.Spare84 := 0;
   Program2.Spare85 := 0;
   Program2.Spare86 := 0;
   Program2.Spare87 := 0;
   Program2.Spare88 := 0;
   Program2.Overlap8_9 := 0;
   Program2.Height9 := 0;
   Program2.Landmark9 := FALSE;
   Program2.Lifter9 := FALSE;
   Program2.SpareBit1H9 := FALSE;
   Program2.Airblower9 := FALSE;
   Program2.NextStep9 := TRUE;
   Program2.PressureP9 := FALSE;
   Program2.SpareByte2H9 := 16#00;
   Program2.Revolution9 := 1;
   Program2.RopeUnit9_1 := 16#01;
   Program2.RopeUnit9_2 := 16#01;
   Program2.FilmForce9 := 0;
   Program2.FilmPrestretch9 := 100;
   Program2.Spare3H9 := 0;
   Program2.Spare89 := 0;
   Program2.Spare90 := 0;
   Program2.Spare91 := 0;
   Program2.Spare92 := 0;
   Program2.Spare93 := 0;
   Program2.Overlap9_10 := 0;
   Program2.Height10 := 0;
   Program2.Landmark10 := FALSE;
   Program2.Lifter10 := FALSE;
   Program2.SpareBit1H10 := FALSE;
   Program2.Airblower10 := FALSE;
   Program2.NextStep10 := FALSE;
   Program2.PressureP10 := FALSE;
   Program2.SpareByte2H10 := 16#00;
   Program2.Revolution10 := 1;
   Program2.RopeUnit10_1 := 16#01;
   Program2.RopeUnit10_2 := 16#01;
   Program2.FilmForce10 := 0;
   Program2.FilmPrestretch10 := 100;
   Program2.Spare3H10 := 0;
   Program2.Spare94 := 0;
   Program2.Spare95 := 0;
   Program2.Spare96 := 0;
   Program2.Spare97 := 0;
   Program2.Spare98 := 0;
   Program2.Overlap10_11 := 0;
   Program2.Height11 := 0;
   Program2.Landmark11 := FALSE;
   Program2.Lifter11 := FALSE;
   Program2.SpareBit1H11 := FALSE;
   Program2.Airblower11 := FALSE;
   Program2.NextStep11 := TRUE;
   Program2.PressureP11 := FALSE;
   Program2.SpareByte2H11 := 16#00;
   Program2.Revolution11 := 1;
   Program2.RopeUnit11_1 := 16#01;
   Program2.RopeUnit11_2 := 16#01;
   Program2.FilmForce11 := 0;
   Program2.FilmPrestretch11 := 100;
   Program2.Spare3H11 := 0;
   Program2.Spare99 := 0;
   Program2.Spare100 := 0;
   Program2.Spare101 := 0;
   Program2.Spare102 := 0;
   Program2.Spare103 := 0;
   Program2.Overlap11_12 := 0;
   Program2.Height12 := 0;
   Program2.Landmark12 := FALSE;
   Program2.Lifter12 := FALSE;
   Program2.SpareBit1H12 := FALSE;
   Program2.Airblower12 := FALSE;
   Program2.NextStep12 := FALSE;
   Program2.PressureP12 := FALSE;
   Program2.SpareByte2H12 := 16#00;
   Program2.Revolution12 := 1;
   Program2.RopeUnit12_1 := 16#01;
   Program2.RopeUnit12_2 := 16#01;
   Program2.FilmForce12 := 0;
   Program2.FilmPrestretch12 := 100;
   Program2.Spare3H12 := 0;
   Program2.Spare104 := 0;
   Program2.Spare105 := 0;
   Program2.Spare106 := 0;
   Program2.Spare107 := 0;
   Program2.Spare108 := 0;
END_DATA_BLOCK

DATA_BLOCK "DB24_AlarmDisplay"   // DB24
{ S7_Optimized_Access := 'FALSE' }
AUTHOR : Robopac
VERSION : 0.0
// stored: AutoNumber false, IsOnlyStoredInLoadMemory false, IsWriteProtectedInAS false
   VAR RETAIN
      Alarm1 : Byte := 16#00;   // Alarm byte 1
      Alarm2 : Byte := 16#00;   // Alarm byte 2
      Alarm3 : Byte := 16#00;   // Alarm byte 3
      Alarm4 : Byte := 16#00;   // Alarm byte 4
      Alarm5 : Byte := 16#00;   // Alarm byte 5
      Alarm6 : Byte := 16#00;   // Alarm byte 6
      Alarm7 : Byte := 16#00;   // Alarm byte 7
      Alarm8 : Byte := 16#00;   // Alarm byte 8
      Alarm9 : Byte := 16#00;   // Alarm byte 9
      Alarm10 : Byte := 16#00;   // Alarm byte 10
      Alarm11 : Byte := 16#00;   // Alarm byte 11
      Alarm12 : Byte := 16#00;   // Alarm byte 12
      Alarm13 : Byte := 16#00;   // Alarm byte 13
      Alarm14 : Byte := 16#00;   // Alarm byte 14
      Alarm15 : Byte := 16#00;   // Alarm byte 15
      Alarm16 : Byte := 16#00;   // Alarm byte 16
      Alarm17 : Byte := 16#00;   // Alarm byte 17
      Alarm18 : Byte := 16#00;   // Alarm byte 18
      Alarm19 : Byte := 16#00;   // Alarm byte 19
      Alarm20 : Byte := 16#00;   // Alarm byte 20
      Alarm21 : Byte := 16#00;   // Alarm byte 21
      Alarm22 : Byte := 16#00;   // Alarm byte 22
      Alarm23 : Byte := 16#00;   // Alarm byte 23
      Alarm24 : Byte := 16#00;   // Alarm byte 24
      Alarm25 : Byte := 16#00;   // Alarm byte 25
      Alarm26 : Byte := 16#00;   // Alarm byte 26
      Alarm27 : Byte := 16#00;   // Alarm byte 27
      Alarm28 : Byte := 16#00;   // Alarm byte 28
      Alarm29 : Byte := 16#00;   // Alarm byte 29
      Alarm30 : Byte := 16#00;   // Alarm byte 30
      Alarm31 : Byte := 16#00;   // Alarm byte 31
      Alarm32 : Byte := 16#00;   // Alarm byte 32
      Alarm33 : Byte := 16#00;   // Alarm byte 33
      Alarm34 : Byte := 16#00;   // Alarm byte 34
      Alarm35 : Byte := 16#00;   // Alarm byte 35
      Alarm36 : Byte := 16#00;   // Alarm byte 36
      Alarm37 : Byte := 16#00;   // Alarm byte 37
      Alarm38 : Byte := 16#00;   // Alarm byte 38
      Alarm39 : Byte := 16#00;   // Alarm byte 39
      Alarm40 : Byte := 16#00;   // Alarm byte 40
      AckAlarm1 : Byte := 16#00;   // Alarm acknowledge for byte 1
      AckAlarm2 : Byte := 16#00;   // Alarm acknowledge for byte 2
      AckAlarm3 : Byte := 16#00;   // Alarm acknowledge for byte 3
      AckAlarm4 : Byte := 16#00;   // Alarm acknowledge for byte 4
      AckAlarm5 : Byte := 16#00;   // Alarm acknowledge for byte 5
      AckAlarm6 : Byte := 16#00;   // Alarm acknowledge for byte 6
      AckAlarm7 : Byte := 16#00;   // Alarm acknowledge for byte 7
      AckAlarm8 : Byte := 16#00;   // Alarm acknowledge for byte 8
      AckAlarm9 : Byte := 16#00;   // Alarm acknowledge for byte 9
      AckAlarm10 : Byte := 16#00;   // Alarm acknowledge for byte 10
      AckAlarm11 : Byte := 16#00;   // Alarm acknowledge for byte 11
      AckAlarm12 : Byte := 16#00;   // Alarm acknowledge for byte 12
      AckAlarm13 : Byte := 16#00;   // Alarm acknowledge for byte 13
      AckAlarm14 : Byte := 16#00;   // Alarm acknowledge for byte 14
      AckAlarm15 : Byte := 16#00;   // Alarm acknowledge for byte 15
      AckAlarm16 : Byte := 16#00;   // Alarm acknowledge for byte 16
      AckAlarm17 : Byte := 16#00;   // Alarm acknowledge for byte 17
      AckAlarm18 : Byte := 16#00;   // Alarm acknowledge for byte 18
      AckAlarm19 : Byte := 16#00;   // Alarm acknowledge for byte 19
      AckAlarm20 : Byte := 16#00;   // Alarm acknowledge for byte 20
      AckAlarm21 : Byte := 16#00;   // Alarm acknowledge for byte 21
      AckAlarm22 : Byte := 16#00;   // Alarm acknowledge for byte 22
      AckAlarm23 : Byte := 16#00;   // Alarm acknowledge for byte 23
      AckAlarm24 : Byte := 16#00;   // Alarm acknowledge for byte 24
      AckAlarm25 : Byte := 16#00;   // Alarm acknowledge for byte 25
      AckAlarm26 : Byte := 16#00;   // Alarm acknowledge for byte 26
      AckAlarm27 : Byte := 16#00;   // Alarm acknowledge for byte 27
      AckAlarm28 : Byte := 16#00;   // Alarm acknowledge for byte 28
      AckAlarm29 : Byte := 16#00;   // Alarm acknowledge for byte 29
      AckAlarm30 : Byte := 16#00;   // Alarm acknowledge for byte 30
      AckAlarm31 : Byte := 16#00;   // Alarm acknowledge for byte 31
      AckAlarm32 : Byte := 16#00;   // Alarm acknowledge for byte 32
      AckAlarm33 : Byte := 16#00;   // Alarm acknowledge for byte 33
      AckAlarm34 : Byte := 16#00;   // Alarm acknowledge for byte 34
      AckAlarm35 : Byte := 16#00;   // Alarm acknowledge for byte 35
      AckAlarm36 : Byte := 16#00;   // Alarm acknowledge for byte 36
      AckAlarm37 : Byte := 16#00;   // Alarm acknowledge for byte 37
      AckAlarm38 : Byte := 16#00;   // Alarm acknowledge for byte 38
      AckAlarm39 : Byte := 16#00;   // Alarm acknowledge for byte 39
      AckAlarm40 : Byte := 16#00;   // Alarm acknowledge for byte 40
   END_VAR
BEGIN
END_DATA_BLOCK

DATA_BLOCK "DB252_ProgramGreyBar"   // DB252
{ S7_Optimized_Access := 'FALSE' }
VERSION : 0.1
// stored: AutoNumber false, IsOnlyStoredInLoadMemory false, IsWriteProtectedInAS false
   VAR RETAIN
      Height { ExternalAccessible := 'False'; ExternalVisible := 'False'; ExternalWritable := 'False'; S7_SetPoint := 'True'} : Array[1..13] of "ProgramDataGreyBar";
   END_VAR
BEGIN
   Height[1..2].Overlap := 0;
   Height[3..4].Overlap := 100;
   Height[5..13].Overlap := 0;
   Height[1].Height := 130;
   Height[2].Height := 50;
   Height[3].Height := -50;
   Height[4].Height := 100;
   Height[5].Height := 50;
   Height[6..13].Height := 0;
   Height[1..2].Landmark := FALSE;
   Height[3].Landmark := TRUE;
   Height[4..13].Landmark := FALSE;
   Height[1..13].Lifter := FALSE;
   Height[1..13].SpareBit1 := FALSE;
   Height[1..5].Airblower := TRUE;
   Height[6..13].Airblower := FALSE;
   Height[1..4].NextStep := TRUE;
   Height[5..13].NextStep := FALSE;
   Height[1..4].PressureP := TRUE;
   Height[5..13].PressureP := FALSE;
   Height[1..13].SpareByte1 := 16#00;
   Height[1..2].Revolution := 1;
   Height[3].Revolution := 2;
   Height[4].Revolution := 3;
   Height[5].Revolution := 1;
   Height[6..13].Revolution := 0;
   Height[1..3].RopeUnitUpper := 16#01;
   Height[4].RopeUnitUpper := 16#02;
   Height[5].RopeUnitUpper := 16#01;
   Height[6..13].RopeUnitUpper := 16#00;
   Height[1..3].RopeUnitLower := 16#01;
   Height[4].RopeUnitLower := 16#02;
   Height[5].RopeUnitLower := 16#01;
   Height[6..13].RopeUnitLower := 16#00;
   Height[1].FilmForce := 5;
   Height[2].FilmForce := 20;
   Height[3..5].FilmForce := 30;
   Height[6..13].FilmForce := 0;
   Height[1..5].FilmPrestretch := 200;
   Height[6..13].FilmPrestretch := 0;
   Height[1..13].SpareWord1 := 0;
   Height[1..13].SpareWord2 := 0;
   Height[1..13].SpareWord3 := 0;
   Height[1..2].SpareWord4 := 0;
   Height[3].SpareWord4 := 380;
   Height[4..13].SpareWord4 := 0;
   Height[1..2].SpareWord5 := 0;
   Height[3].SpareWord5 := 2800;
   Height[4..13].SpareWord5 := 0;
   Height[1..13].SpareWord6 := 0;
END_DATA_BLOCK

DATA_BLOCK "DB25_Display"   // DB25
{ S7_Optimized_Access := 'FALSE' }
AUTHOR : Robopac
VERSION : 0.0
// stored: AutoNumber false, IsOnlyStoredInLoadMemory false, IsWriteProtectedInAS false
   VAR RETAIN
      dbw0 : Int := 2;   // Command area 1 (Display Esa)
      dbw2 : Int := 0;   // Command area 2 (Display Esa)
      dbw4 : Int := 0;   // Command area 3 (Display Esa)
      dbw6 : Int := 0;   // Command area 4 (Display Esa)
      dbb8 : Byte := 16#00;   // Status area 1 (Display Esa)
      dbx9_0 : Bool := FALSE;   // Status area 1 (Display Esa): Watchdog
      dbx9_1 : Bool := FALSE;   // Status area 1 (Display Esa): Display in editing
      dbw10 : Int := 0;   // Status area 2 (Display Esa)
      dbw12 : Int := 1;   // Status area 3 Current Page (Display Esa)
      dbw14 : Int := 0;   // Status area 4 (Display Esa)
      dbw16 : Int := 0;
      dbw18 : Int := 2;   // Active program on grey bar
      dbx20_0 : Bool := FALSE;   // Grey bar data 1: Wrapping excluded
      dbx20_1 : Bool := TRUE;   // Grey bar data 1: Wrapping included
      dbx20_2 : Bool := FALSE;   // Grey bar data 1: Wrapping included + Top
      dbx20_3 : Bool := TRUE;   // Grey bar data 1: Pressure plate included/excluded
      dbx20_4 : Bool := FALSE;   // Grey bar data 1: Lifter plate included/excluded
      dbx20_5 : Bool := FALSE;
      dbx20_6 : Bool := FALSE;
      dbx20_7 : Bool := FALSE;
      dbx21_0 : Bool := FALSE;   // Grey bar data 1: Step 1_6 or 7_12(1) shown
      dbx21_1 : Bool := FALSE;   // Grey bar data 1: Data loaded for grey bar
      dbx21_2 : Bool := FALSE;
      dbx21_3 : Bool := FALSE;
      dbx21_4 : Bool := FALSE;
      dbx21_5 : Bool := FALSE;
      dbx21_6 : Bool := FALSE;
      dbx21_7 : Bool := FALSE;
      dbw22 : Int := 5;   // Grey bar data 2: Quote active
      dbw24 : Int := 2;   // Grey bar data 3:
      dbw26 : Int := 0;   // Grey bar data 4:
      dbw28 : Int := 0;   // Grey bar data 5:
      dbw30 : Int := 1;   // Copy of current page
      dbx32_0 : Bool := FALSE;   // Program bit: Load data from data table to display area
      dbx32_1 : Bool := FALSE;   // Program bit: Save data from display area to data table
      dbx32_2 : Bool := FALSE;   // Program bit: Blink load button
      dbx32_3 : Bool := FALSE;   // Program bit: Blink load button
      dbx32_4 : Bool := FALSE;   // Program bit: Blink save button
      dbx32_5 : Bool := FALSE;   // Program bit: Blink save button
      dbx32_6 : Bool := FALSE;   // Program data modified on display
      dbx32_7 : Bool := FALSE;
      dbx33_0 : Bool := FALSE;   // Return to page 1 after 3 minutes
      dbx33_1 : Bool := FALSE;   // Exit from alarm page
      dbx33_2 : Bool := FALSE;   // Support for display communication timeout
      dbx33_3 : Bool := FALSE;   // Jump to no password page
      dbx33_4 : Bool := FALSE;   // Support memory for pressure plate grey bar
      dbx33_5 : Bool := FALSE;   // Support memory for lifter grey bar
      dbx33_6 : Bool := FALSE;   // Display on sysdata or maintenance page
      dbx33_7 : Bool := FALSE;   // Request to reset the counter for wrapped pallet (Micrologix)
      dbw34 : Int := 1;   // Copy of program to be shown on display
      dbw36 : Int := 18;   // Old page used on alarm exit
      dbw38 : Int := 5;   // Support memory for quote active
      dbx40_0 : Bool := FALSE;   // Pallet on conveyor bit: Conveyor CM
      dbx40_1 : Bool := FALSE;   // Pallet on conveyor bit: Conveyor pos.1 (infeed)
      dbx40_2 : Bool := TRUE;   // Pallet on conveyor bit: Conveyor pos.2 (outfeed)
      dbx40_3 : Bool := FALSE;   // Pallet on conveyor bit:
      dbx40_4 : Bool := TRUE;   // Pallet on conveyor bit:
      dbx40_5 : Bool := FALSE;   // Pallet on conveyor bit:
      dbb41 : Byte := 16#00;   // Pallet on rotoplat conveyor byte: 0 empty, 1 pallet, 2 empty 90, 3 pallet 90
      dbw42 : Int := 0;   // Command area 1 (Display Siemens TP) -
      dbw44 : Word := 16#0000;   // Command area 2 (Display Siemens TP)
      dbw46 : Word := 16#0000;   // Command area 3 (Display Siemens TP)
      dbw48 : Word := 16#0000;   // Command area 4 (Display Siemens TP)
      dbb50 : Byte := 16#00;   // Status area (Display Siemens TP):
      dbx51_0 : Bool := TRUE;   // Status area (Display Siemens TP): Start bit
      dbx51_1 : Bool := FALSE;   // Status area (Display Siemens TP): Display offline/online
      dbx51_2 : Bool := FALSE;   // Status area (Display Siemens TP): Watchdog
      dbw52 : Word := 16#0001;   // Status area (Display Siemens TP): Current page type
      dbw54 : Int := 1;   // Status area (Display Siemens TP): Current page number
      dbw56 : Word := 16#0000;   // Status area (Display Siemens TP): Reserved
      dbw58 : Word := 16#0001;   // Status area (Display Siemens TP): Current object number
      dbw60 : Word := 16#0000;   // Status area (Display Siemens TP): Reserved
      ProgQuoteQX : Int := 0;   // Multiplex Wincc - Program data
      ProgBitQX : Int := 4;   // Multiplex Wincc - Program data
      ProgQuotaQX : Int := 2;   // Multiplex Wincc - Program data
      ProgGiriQX : Int := 6;   // Multiplex Wincc - Program data
      ProgSovrappQX : Int := 0;   // Multiplex Wincc - Program data
      ProgStringifasciaQX : Int := 8;   // Multiplex Wincc - Program data
      ProgTiroFilmQX : Int := 10;   // Multiplex Wincc - Program data
      ProgPrestiroFilmQX : Int := 12;   // Multiplex Wincc - Program data
      ProgStringifascia2QX : Int := 9;   // Multiplex Wincc - Program data
      dbw80 : Int := 3;   // Multiplex Wincc - Program data
      dbw82 : Int := 0;
      dbw84 : Int := 0;
      dbw86 : Int := 0;
      dbw88 : Int := 0;
      dbw90 : Int := 0;
      dbw92 : Int := 0;
      dbw94 : Int := 0;
      dbw96 : Int := 0;
      dbw98 : Int := 130;
   END_VAR
BEGIN
END_DATA_BLOCK

DATA_BLOCK "DB26"   // DB26
{ S7_Optimized_Access := 'FALSE' }
VERSION : 0.1
// stored: AutoNumber false, IsOnlyStoredInLoadMemory false, IsWriteProtectedInAS false
   VAR RETAIN
      Dbd0 : Real := 0.0;   // Valore massimo di scalatura dell'uscita = 32000
      Dbd4 : Real := 0.0;   // Valore minimo di scalatura dell'uscita = 0.0
      Dbd8 : Real := 0.0;   // Valore massimo di scalatura della parola di ingresso = 100-%tiro
      Dbd12 : Real := 0.0;   // Valore minimo di scalatura della parola di ingresso analogico = 0.0
      Dbd16 : DInt := 0;   // valore di prestiro impostato sul display convertito a 32 bit
      Dbd20 : Real := 0.0;   // valore di prestiro impostato sul display a 32 bit convertito in virgola mobile
      Dbd24 : Real := 0.0;   // Differenza fra valore massimo di scal.e valore minimo di scal.all'uscita
      Dbd28 : Real := 0.0;   // Differenza fra valore massimo di scal.e valore minimo di scal.all'input analogi
      Dbd32 : Real := 0.0;   // differenza fra dbd20 e dbd 12
      Dbd36 : Real := 0.0;
      Dbd40 : Real := 0.0;
      Dbd44 : Real := 0.0;
      Dbw48 : Int := 0;
      Dbw50 : Int := 200;   // valore di prestiro impostato sul display a 16 bit
      Dbw52 : Int := 0;   // valore di tiro impostato sul display a 16 bit
      Dbd54 : DInt := 0;
      Dbd58 : DInt := 0;
      Dbd62 : Real := 0.0;
      Dbd66 : Real := 0.0;
      Dbd70 : Real := 0.0;
      Dbd74 : Real := 0.0;
      Dbd78 : Real := 0.0;
      Dbd82 : DInt := 0;
      Dbw86 : Int := 0;   // valore di tiro impostato sul display a 16 bit per ciclo taglio
      Dbw88 : Int := 5;   // valore di tiro impostato sul display a 16 bit per ciclo avvolgitura
      Dbw90 : Int := 0;   // valore di tiro impostato sul display a 16 bit per inizio ciclo
      Dbw92 : Int := 0;
      Dbw94 : Int := 0;
      Dbw96 : Int := 0;
      Dbw98 : Int := 0;
      Dbw100 : Int := 0;
      Dbw102 : Int := 0;
      Dbw104 : Int := 0;
      Dbw106 : Int := 0;
      Dbw108 : Int := 0;
      Dbw110 : Int := 0;
      Dbw112 : Int := 0;
      Dbw114 : Int := 0;
      Dbw116 : Int := 0;
   END_VAR
BEGIN
END_DATA_BLOCK

DATA_BLOCK "DB321_PID_M20"   // DB321
TITLE = PID
{ S7_Optimized_Access := 'FALSE' }
VERSION : 0.1
// stored: AutoNumber false, IsOnlyStoredInLoadMemory false, IsWriteProtectedInAS false
   VAR RETAIN
      PID { S7_SetPoint := 'True'} : "M20";
   END_VAR
BEGIN
   PID.M20_P00 := 0;
   PID.M20_P01 := 70;
   PID.M20_P02 := 15;
   PID.M20_P03 := 0;
   PID.M20_P04 := 60;
   PID.M20_P05 := 7;
   PID.M20_P06 := 200;
   PID.M20_P07 := 200;
   PID.M20_P08 := 65;
   PID.M20_P09 := 240;
   PID.M20_P10 := 100;
   PID.M20_P11 := 128;
   PID.M20_P12 := 10;
   PID.M20_P13 := 0;
   PID.M20_P14 := 6;
   PID.M20_P15 := 50;
   PID.M20_P20 := 0;
   PID.M20_P21 := 0;
   PID.M20_P22 := 0;
   PID.M20_P23 := 0;
   PID.M20_P24 := 0;
   PID.M20_P25 := 0;
END_DATA_BLOCK

DATA_BLOCK "DB91_NetDB"   // DB91
{ S7_Optimized_Access := 'FALSE' }
VERSION : 0.1
// stored: AutoNumber false, IsOnlyStoredInLoadMemory false, IsWriteProtectedInAS false
   VAR RETAIN
      In_livebit : Bool := FALSE;   // set this bit to TRUE
      spare1 : Bool := FALSE;
      spare2 : Bool := FALSE;
      spare3 : Bool := FALSE;
      spare4 : Bool := FALSE;
      spare5 : Bool := FALSE;
      spare6 : Bool := FALSE;
      spare7 : Bool := FALSE;
      IN_PRI : Bool := FALSE;   // Pallet ready in infeed
      IN_RRO : Bool := FALSE;   // Ready to receive in outfeed
      IN_ETO : Bool := FALSE;   // End of transfer in outfeed
      IN_EXC : Bool := FALSE;   // Wrapping excluded signal
      IN_ResetPartial : Bool := FALSE;   // Reset partial wrapped counter
      IN_spare5 : Bool := FALSE;
      IN_spare6 : Bool := FALSE;
      IN_spare7 : Bool := FALSE;
      IN_Program : Byte := 16#00;   // Program selection byte 1-15 (0 excluded)
      OUT_RRI : Bool := FALSE;   // Ready to receive in infeed signal
      OUT_ETI : Bool := FALSE;   // End of transfer in infeed signal
      OUT_PRO : Bool := FALSE;   // Pallet ready in outfeed signal
      OUT_spare3 : Bool := FALSE;
      OUT_spare4 : Bool := FALSE;
      OUT_spare5 : Bool := FALSE;
      OUT_spare6 : Bool := FALSE;
      Out_LiveBit : Bool := FALSE;   // This bit always TRUE
      spare_word : Word := 16#0000;
      MachineStatus : Word := 16#0000;
      WorkedHours : DWord := 16#0000_0000;
      PalletWrapped : DWord := 16#0000_0000;
      PartialWrapped : DWord := 16#0000_0000;
      VD2300 : DWord := 16#0000_0000;
      VD2304 : DWord := 16#0000_0000;
      VD2308 : DWord := 16#0000_0000;
      VD2312 : DWord := 16#0000_0000;
      VD2316 : DWord := 16#0000_0000;
      VD2320 : DWord := 16#0000_0000;
      VD2324 : DWord := 16#0000_0000;
      VW2328 : Word := 16#0000;
   END_VAR
BEGIN
END_DATA_BLOCK

DATA_BLOCK "Inverter_Alarms"   // DB209
TITLE = Inverter Alarms
{ S7_Optimized_Access := 'FALSE' }
VERSION : 0.1
// stored: AutoNumber false, IsOnlyStoredInLoadMemory false, IsWriteProtectedInAS false
   VAR
      U201_alarm : Word := 16#0000;
      U221_alarm : Word := 16#0000;
      U241_alarm : Word := 16#0000;
      U261_alarm : Word := 16#0000;
      U321_alarm : Word := 16#0000;
   END_VAR
BEGIN
END_DATA_BLOCK

DATA_BLOCK "MB_REG1"   // DB201
{ S7_Optimized_Access := 'FALSE' }
VERSION : 0.1
// stored: AutoNumber false, IsOnlyStoredInLoadMemory false, IsWriteProtectedInAS false
   VAR RETAIN
      AD_R : UDInt := 40001;
      LN_R : UInt := 5;
      AD_W : UDInt := 0;
      LN_W : UInt := 0;
      A08R : Struct   // Prestiro_READ
         REG_0 : Int := 227;   // REG_CELLA
         REG_1 : Int := 24;   // REG_INPUT
         REG_2 : Int := 106;   // REG_VERSIONE
         REG_3 : Int := 0;   // REG_ENC1
         REG_4 : Int := 0;   // REG_ENC2
      END_STRUCT;
      A08W : Struct   // Prestiro_WRITE
         REG_5 : Int := 0;   // REG_OUTPUT1
         REG_6 : Int := 0;   // REG_OUTPUT2
         REG_7 : Int := 0;   // REG_OUTPUT3
         REG_8 : Int := 0;   // REG_ENCDIR
         REG_9 : Int := 0;
      END_STRUCT;
      SER : Struct   // Cordonatore_READ
         REG_10 : Int := 12337;
         REG_11 : Int := 12598;
         REG_12 : Int := 18480;
         REG_13 : Int := 12336;
         REG_14 : Int := 12592;
         REG_15 : Int := 0;
         REG_16 : Int := 0;
         REG_17 : Int := 0;
         REG_18 : Int := 0;
         REG_19 : Int := 0;
      END_STRUCT;
   END_VAR
BEGIN
END_DATA_BLOCK

DATA_BLOCK "DB01_Osr"   // DB1
{ S7_Optimized_Access := 'FALSE' }
AUTHOR : Robopac
VERSION : 0.0
// stored: AutoNumber false, IsOnlyStoredInLoadMemory false, IsWriteProtectedInAS false
   VAR RETAIN
      osr1 : Bool := TRUE;   // Used
      osr2 : Bool := FALSE;   // Used
      osr3 : Bool := FALSE;   // Used
      osr4 : Bool := FALSE;   // Used
      osr5 : Bool := FALSE;   // Used
      osr6 : Bool := TRUE;   // Used
      osr7 : Bool := TRUE;   // Used
      osr8 : Bool := FALSE;   // Used
      osr9 : Bool := TRUE;   // Used
      osr10 : Bool := FALSE;   // Used
      osr11 : Bool := FALSE;   // Used
      osr12 : Bool := FALSE;   // Used
      osr13 : Bool := FALSE;   // Used
      osr14 : Bool := FALSE;   // Used
      osr15 : Bool := TRUE;   // Used
      osr16 : Bool := FALSE;   // Used
      osr17 : Bool := TRUE;   // Used
      osr18 : Bool := TRUE;   // Used
      osr19 : Bool := TRUE;   // Used
      osr20 : Bool := TRUE;   // Used
      osr21 : Bool := TRUE;   // Used
      osr22 : Bool := TRUE;   // Used
      osr23 : Bool := FALSE;   // Used
      osr24 : Bool := FALSE;   // Used
      osr25 : Bool := FALSE;   // Used
      osr26 : Bool := FALSE;   // Used
      osr27 : Bool := FALSE;   // Used
      osr28 : Bool := FALSE;   // Used
      osr29 : Bool := FALSE;   // Used
      osr30 : Bool := TRUE;   // Used
      osr31 : Bool := TRUE;   // Used
      osr32 : Bool := TRUE;   // Used
      osr33 : Bool := TRUE;   // Used
      osr34 : Bool := TRUE;   // Used
      osr35 : Bool := FALSE;   // Used
      osr36 : Bool := FALSE;   // Used
      osr37 : Bool := TRUE;
      osr38 : Bool := FALSE;   // Used
      osr39 : Bool := TRUE;   // Used
      osr40 : Bool := FALSE;   // Used
      osr41 : Bool := TRUE;   // Used
      osr42 : Bool := TRUE;
      osr43 : Bool := TRUE;
      osr44 : Bool := FALSE;
      osr45 : Bool := FALSE;   // Used
      osr46 : Bool := FALSE;   // Used
      osr47 : Bool := FALSE;
      osr48 : Bool := FALSE;
      osr49 : Bool := FALSE;
      osr50 : Bool := TRUE;
      osr51 : Bool := FALSE;
      osr52 : Bool := TRUE;
      osr53 : Bool := FALSE;
      osr54 : Bool := FALSE;
      osr55 : Bool := FALSE;
      osr56 : Bool := TRUE;
      osr57 : Bool := FALSE;
      osr58 : Bool := FALSE;
      osr59 : Bool := FALSE;
      osr60 : Bool := TRUE;
      osr61 : Bool := FALSE;
      osr62 : Bool := FALSE;
      osr63 : Bool := FALSE;
      osr64 : Bool := FALSE;
      osr65 : Bool := FALSE;
      osr66 : Bool := FALSE;
      osr67 : Bool := TRUE;
      osr68 : Bool := FALSE;
      osr69 : Bool := TRUE;
      osr70 : Bool := FALSE;
      osr71 : Bool := FALSE;
      osr72 : Bool := FALSE;
      osr73 : Bool := FALSE;
      osr74 : Bool := TRUE;
      osr75 : Bool := TRUE;
      osr76 : Bool := FALSE;
      osr77 : Bool := TRUE;
      osr78 : Bool := TRUE;
      osr79 : Bool := FALSE;
      osr80 : Bool := FALSE;
      osr81 : Bool := FALSE;   // Used
      osr82 : Bool := FALSE;   // Used
      osr83 : Bool := FALSE;
      osr84 : Bool := FALSE;
      osr85 : Bool := FALSE;
      osr86 : Bool := FALSE;
      osr87 : Bool := FALSE;
      osr88 : Bool := TRUE;
      osr89 : Bool := FALSE;
      osr90 : Bool := FALSE;   // Used
      osr91 : Bool := FALSE;
      osr92 : Bool := FALSE;
      osr93 : Bool := TRUE;
      osr94 : Bool := TRUE;
      osr95 : Bool := TRUE;
      osr96 : Bool := TRUE;
   END_VAR
BEGIN
END_DATA_BLOCK

DATA_BLOCK "DB03_Machine"   // DB3
{ S7_Optimized_Access := 'FALSE' }
AUTHOR : Robopac
VERSION : 0.0
// stored: AutoNumber false, IsOnlyStoredInLoadMemory false, IsWriteProtectedInAS false
   VAR RETAIN
      dbx0_0 : Bool := FALSE;   // Enable the arm rotation revolution counter
      dbx0_1 : Bool := FALSE;   // High pressure on prestretch roller dancer
      dbx0_2 : Bool := FALSE;   // One arm revolution done support memory
      dbx0_3 : Bool := FALSE;   // One arm revolution done
      dbx0_4 : Bool := FALSE;   // Support memory for revolution counter
      dbx0_5 : Bool := FALSE;   // Support memory for 10% prestretch carriage
      dbx0_6 : Bool := FALSE;
      dbx0_7 : Bool := FALSE;   // Support memory for arm rotation speed recorded
      dbb1 : Byte := 16#00;
      MachineExc : Bool := FALSE;   // Wrapping excluded
      MachineInc : Bool := FALSE;   // Wrapping included
      dbb3 : Byte := 16#00;
      dbx4_0 : Bool := FALSE;   // Memory to silent acoustic signal on alarm
      dbx4_1 : Bool := FALSE;
      dbx4_2 : Bool := FALSE;   // Condition to check all out of positon alarm
      dbx4_3 : Bool := FALSE;   // Condition for manual operation
      dbx4_4 : Bool := FALSE;   // All units are ready for automatic cycle
      dbx4_5 : Bool := FALSE;
      dbx4_6 : Bool := FALSE;   // Data for next ring height loaded
      dbx4_7 : Bool := FALSE;   // Data for next ring height loaded
      dbx5_0 : Bool := FALSE;   // Wrapping cycle: Next step is cut and pallet unload
      dbx5_1 : Bool := FALSE;   // Wrapping cycle: Next step is cut and new spool carriage height
      dbx5_2 : Bool := FALSE;   // Wrapping cycle: Next step is new spool carriage height
      dbx5_3 : Bool := FALSE;   // Wrapping cycle: After this step top waterproof
      dbx5_4 : Bool := FALSE;   // Wrong data program for the pallet on the machine
      dbx5_5 : Bool := FALSE;   // Closing upper(double) rope unit
      dbx5_6 : Bool := FALSE;   // Closing single or lower(double) rope unit
      dbx5_7 : Bool := FALSE;   // Memory for timeout enable
      dbx6_0 : Bool := FALSE;   // Memory to exclude infeed safety barrier
      dbx6_1 : Bool := FALSE;   // Memory to exclude outfeed safety barrier
      dbx6_2 : Bool := FALSE;   // Memory to exclude infeed safety barrier
      dbx6_3 : Bool := FALSE;   // Memory to exclude infeed safety barrier
      dbx6_4 : Bool := FALSE;   // Memory to exclude outfeed safety barrier
      dbx6_5 : Bool := FALSE;   // Memory to exclude outfeed safety barrier
      dbx6_6 : Bool := FALSE;
      dbx6_7 : Bool := FALSE;
      dbx7_0 : Bool := FALSE;   // Pressure plate excluded for low pallet
      dbx7_1 : Bool := FALSE;
      dbx7_2 : Bool := FALSE;   // Support memory to check rotation speed
      dbx7_3 : Bool := FALSE;   // Support memory to check spool carriage speed
      dbx7_4 : Bool := FALSE;   // Used by S7-200
      dbx7_5 : Bool := FALSE;   // Machine in wrapping cycle
      dbx7_6 : Bool := FALSE;   // Support memory to refresh pallet per hour value
      dbx7_7 : Bool := FALSE;
      dbb8 : Byte := 16#00;
      TopExc : Bool := FALSE;   // Top excluded
      TopBefore : Bool := FALSE;   // Top included before wrapping beginning
      TopWaterP : Bool := FALSE;   // Top included waterproof
      dbw10 : Int := 0;
      dbw12 : Int := 0;   // Counter for revolution on running spool carriage height
      dbw14 : Int := 0;   // Counter for revolution on welder contrast
      dbw16 : Int := 0;   // Counter for revolution of deceleration
      dbw18 : Int := 0;
      dbw20 : Int := 0;   // Active program for multiprogram (Display)
      dbw22 : Int := 0;   // Selected program for multiprogram (Display)
      dbw24 : Int := 0;   // Program to be shown on data program page (Display)
      dbw26 : Int := 0;   // Program selection by external signal
      dbw28 : Int := 0;   // Program selection by external signal
      dbw30 : Int := 0;   // Support memory for data transfer
      dbw32 : Int := 0;   // Arm rotation speed recorded (rpm*10)
      dbw34 : Int := 0;   // Required arm rotation speed recorded (%*10)
      dbw36 : Int := 0;
      dbw38 : Int := 0;   // Support memory to evaluate carriage movement speed
      dbw40 : Int := 0;   // Support memory to evaluate carriage movement speed
      dbw42 : Int := 0;   // Spool carriage movement speed mm/sec
      dbw44 : Int := 0;   // table rotation movement speed mm/sec
      dbw46 : Int := 0;   // Arm rotation speed (rpm*10) related to actual required speed
      dbw48 : Int := 0;   // Spool carriage movement speed mm/sec recorded
      dbw50 : Int := 0;
      dbw52 : Int := 0;   // High speed for spool carriage movement (%) recorded from display
      dbw54 : Int := 0;   // upport memory for spool carriage high speed
      dbw56 : Int := 0;   // Spool carriage movement speed used on cycle (mm/sec)
      dbb58 : Byte := 16#00;   // Counter for DAC M20 converter
      dbx59_0 : Bool := FALSE;   // Arm rotation and top carriage speed change for DAC M20
      dbx59_1 : Bool := FALSE;   // Spool carriage speed change for DAC M20
      dbx59_2 : Bool := FALSE;   // Counter for DAC M20 is odd
      dbx59_3 : Bool := FALSE;
      dbx59_4 : Bool := FALSE;
      dbx59_5 : Bool := FALSE;
      dbx59_6 : Bool := FALSE;
      dbx59_7 : Bool := FALSE;
      dbw60 : Int := 0;   // Value for DAC analog output
      dbw62 : Int := 0;
      dbw64 : Int := 0;
      dbw66 : Int := 0;   // Support for running height data transfer
      dbw68 : Int := 0;   // Number of the running spool carriage height
      dbw70 : Int := 0;   // Film overlap for running spool carriage height
      dbw72 : Int := 0;   // Carriage height (mm) for running spool carriage height
      dbx74_0 : Bool := FALSE;   // Landmark (0=Bottom 1=Top) for running spool carriage height
      dbx74_1 : Bool := FALSE;   // Pallet lifter for running spool carriage height (0=Excluded 1=Included)
      dbx74_2 : Bool := FALSE;   // Spare
      dbx74_3 : Bool := FALSE;   // Airblower on film tail for running spool carriage height (0=Exc 1=Inc)
      dbx74_4 : Bool := FALSE;   // Next step for running spool carriage height (0=End 1=Next)
      dbx74_5 : Bool := FALSE;   // Pressure plate for running spool carriage height (0=Excluded 1=Included)
      dbx74_6 : Bool := FALSE;   // Spare
      dbx74_7 : Bool := FALSE;   // Spare
      dbb75 : Byte := 16#00;   // Spare
      dbw76 : Int := 0;   // Revolutions for running spool carriage height
      dbb78 : Byte := 16#00;   // Rope unit for running spool carriage height (1=Excluded 2=Inc 3=Inc during)
      dbb79 : Byte := 16#00;   // Rope unit for running spool carriage height (1=Excluded 2=Inc 3=Inc during)
      dbw80 : Int := 0;   // Film force for running spool carriage height
      dbw82 : Int := 0;   // Film prestretch for running spool carriage height
      dbw84 : Int := 0;   // Delay to open or close upper rope unit for runninh spool carriage height
      dbw86 : Int := 0;   // Delay to open or close lower rope unit for runninh spool carriage height
      dbw88 : Int := 0;   // Spare for running spool carriage height
      dbw90 : Int := 0;   // Spare for running spool carriage height
      dbw92 : Int := 0;   // Spare for running spool carriage height
      dbw94 : Int := 0;   // Spare for running spool carriage height
      dbw96 : Int := 0;
      dbw98 : Int := 0;
   END_VAR
BEGIN
END_DATA_BLOCK

DATA_BLOCK "DB05_SpoolCarriagePos"   // DB5
{ S7_Optimized_Access := 'FALSE' }
AUTHOR : Robopac
VERSION : 0.0
// stored: AutoNumber false, IsOnlyStoredInLoadMemory false, IsWriteProtectedInAS false
   VAR RETAIN
      dbx0_0 : Bool := FALSE;   // Table rotation forward
      dbx0_1 : Bool := FALSE;   // Table rotation backward
      dbx0_2 : Bool := FALSE;   // Table rotation speed: Low
      dbx0_3 : Bool := FALSE;   // Table rotation speed: Middle 1 for top
      dbx0_4 : Bool := FALSE;   // Table rotation speed: Middle 2 for welder contrast
      dbx0_5 : Bool := FALSE;   // Table rotation speed: High
      dbx0_6 : Bool := FALSE;
      dbx0_7 : Bool := FALSE;
      dbx1_0 : Bool := FALSE;   // Spool carriage axis movement upward
      dbx1_1 : Bool := FALSE;   // Spool carriage axis movement downward
      dbx1_2 : Bool := FALSE;   // Spool carriage axis movement inside low speed area
      dbx1_3 : Bool := FALSE;   // Spool carriage axis movement low speed
      dbx1_4 : Bool := FALSE;   // Spool carriage upward
      dbx1_5 : Bool := FALSE;   // Spool carriage downward
      dbx1_6 : Bool := FALSE;
      dbx1_7 : Bool := FALSE;
      dbx2_0 : Bool := FALSE;
      dbx2_1 : Bool := FALSE;   // Support memory for enable (EN) on table rotation and table conveyor inverter
      dbx2_2 : Bool := FALSE;
      dbx2_3 : Bool := FALSE;
      dbx2_4 : Bool := FALSE;
      dbx2_5 : Bool := FALSE;
      dbx2_6 : Bool := FALSE;
      dbx2_7 : Bool := FALSE;
      dbx3_0 : Bool := FALSE;   // Spool carriage: Support for encoder running control
      dbx3_1 : Bool := FALSE;   // Spool carriage: Support for encoder running control alarm
      dbx3_2 : Bool := FALSE;
      dbx3_3 : Bool := FALSE;
      dbx3_4 : Bool := FALSE;
      dbx3_5 : Bool := FALSE;
      dbx3_6 : Bool := FALSE;
      dbx3_7 : Bool := FALSE;
      dbx4_0 : Bool := FALSE;   // Pallet height recording in automatic mode
      dbx4_1 : Bool := FALSE;   // Support memory for pallet height recording
      dbx4_2 : Bool := FALSE;
      dbx4_3 : Bool := FALSE;   // Support memory for pallet height filter
      dbx4_4 : Bool := FALSE;   // Condition for pallet height detected
      dbx4_5 : Bool := FALSE;
      dbx4_6 : Bool := TRUE;   // Carriage in position to rotate in medium to wrap top
      dbx4_7 : Bool := FALSE;
      dbx5_0 : Bool := FALSE;
      dbx5_1 : Bool := FALSE;
      dbx5_2 : Bool := FALSE;
      dbx5_3 : Bool := FALSE;
      dbx5_4 : Bool := TRUE;   // Top wrapped ring position
      dbw6 : Int := 100;   // Spool carriage: Support for movement speed
      dbw8 : Int := 50;   // Spool carriage: Support for movement deceleration
      dbw10 : Int := 100;
      dbw12 : Int := 10199;
      dbw14 : Int := 10306;   // Pallet height on machine conveyor + 300 mm
      dbw16 : Int := 9999;   // Pallet height on machine conveyor
      dbw18 : Int := 9999;   // Pallet height on machine conveyor
      dbw20 : Int := 480;   // Spool carriage height for middle speed on welder contrast
      dbw22 : Int := -2;   // Support memory for pallet height filter
      dbw24 : Int := 0;   // Support memory for pallet height
      dbw26 : Int := -380;   // Spool carriage height for middle speed before top cycle
      dbw28 : Int := 0;
      dbd30 : DInt := -1;   // Spool carriage position: Pulse
      dbw34 : Int := -2;   // Spool carriage position: Top of the spool
      dbw36 : Int := 1782;   // Spool carriage position: Spool carriage all up position
      dbw38 : Int := 50;   // Spool carriage position: Deceleration position for carriage overrun down
      dbw40 : Int := 1732;   // Spool carriage position: Deceleration position for carriage overrun up
      dbd42 : DInt := -1;   // Support for encoder spool carriage running control
      dbw46 : Int := 12;   // Support for encoder spool carriage running control
      dbw48 : Int := 0;
      dbw50 : Int := 0;   // Support memory for machine conveyor speed (%)
      dbw52 : Int := 0;   // Support memory for spool carriage and machine conveyor speed (%)
      dbw54 : Int := 0;   // Support memory for for arm rotation speed (%*10)
      dbw56 : Int := 0;   // Support memory for top carriage forward/backward speed (%*10)
      dbw58 : Int := 0;   // Support memory for top carriage forward/backward and arm rotation speed (%*10)
      dbw60 : Int := 0;
      dbw62 : Int := 0;
      dbw64 : Int := 0;
      dbw66 : Int := 0;
      dbw68 : Int := 0;
      Req1_Start : Bool := FALSE;   // Positioning request 1: Start
      Req2_Start : Bool := FALSE;   // Positioning request 2: Start
      Req3_Start : Bool := FALSE;   // Positioning request 3: Start
      Req4_Start : Bool := FALSE;   // Positioning request 4: Start
      Req5_Start : Bool := FALSE;   // Positioning request 5: Start
      Req6_Start : Bool := FALSE;   // Positioning request 6: Start
      Req7_Start : Bool := FALSE;   // Positioning request 7: Start
      Req8_Start : Bool := FALSE;   // Positioning request 8: Start
      Req9_Start : Bool := FALSE;   // Positioning request 9: Start
      Req10_Start : Bool := FALSE;   // Positioning request 10: Start
      Req1_Dest : Int := 50;   // Positioning request 1: Destination position
      Req2_Dest : Int := 40;   // Positioning request 2: Destination position
      Req3_Dest : Int := -260;   // Positioning request 3: Destination position
      Req4_Dest : Int := 0;   // Positioning request 4: Destination position
      Req1_Fwd : Bool := FALSE;   // Positioning request 1: Axis forward
      Req1_Bkw : Bool := FALSE;   // Positioning request 1: Axis backward
      Req1_Slow : Bool := FALSE;   // Positioning request 1: Axis slow speed
      Req1_Pos : Bool := FALSE;   // Positioning request 1: Axis in position
      Req2_Fwd : Bool := FALSE;   // Positioning request 2: Axis forward
      Req2_Bkw : Bool := FALSE;   // Positioning request 2: Axis backward
      Req2_Slow : Bool := FALSE;   // Positioning request 2: Axis slow speed
      Req2_Pos : Bool := FALSE;   // Positioning request 2: Axis in position
      Req3_Fwd : Bool := FALSE;   // Positioning request 3: Axis forward
      Req3_Bkw : Bool := FALSE;   // Positioning request 3: Axis backward
      Req3_Slow : Bool := FALSE;   // Positioning request 3: Axis slow speed
      Req3_Pos : Bool := FALSE;   // Positioning request 3: Axis in position
      Req4_Fwd : Bool := FALSE;   // Positioning request 4: Axis forward
      Req4_Bkw : Bool := FALSE;   // Positioning request 4: Axis backward
      Req4_Slow : Bool := FALSE;   // Positioning request 4: Axis slow speed
      Req4_Pos : Bool := FALSE;   // Positioning request 4: Axis in position
      Req5_Dest : Int := 0;   // Positioning request 5: Destination position
      Req6_Dest : Int := 0;   // Positioning request 6: Destination position
      Req7_Dest : Int := 0;   // Positioning request 7: Destination position
      Req8_Dest : Int := 0;   // Positioning request 8: Destination position
      Req5_Fwd : Bool := FALSE;   // Positioning request 5: Axis forward
      Req5_Bkw : Bool := FALSE;   // Positioning request 5: Axis backward
      Req5_Slow : Bool := FALSE;   // Positioning request 5: Axis slow speed
      Req5_Pos : Bool := FALSE;   // Positioning request 5: Axis in position
      Req6_Fwd : Bool := FALSE;   // Positioning request 6: Axis forward
      Req6_Bkw : Bool := FALSE;   // Positioning request 6: Axis backward
      Req6_Slow : Bool := FALSE;   // Positioning request 6: Axis slow speed
      Req6_Pos : Bool := FALSE;   // Positioning request 6: Axis in position
      Req7_Fwd : Bool := FALSE;   // Positioning request 7: Axis forward
      Req7_Bkw : Bool := FALSE;   // Positioning request 7: Axis backward
      Req7_Slow : Bool := FALSE;   // Positioning request 7: Axis slow speed
      Req7_Pos : Bool := FALSE;   // Positioning request 7: Axis in position
      Req8_Fwd : Bool := FALSE;   // Positioning request 8: Axis forward
      Req8_Bkw : Bool := FALSE;   // Positioning request 8: Axis backward
      Req8_Slow : Bool := FALSE;   // Positioning request 8: Axis slow speed
      Req8_Pos : Bool := FALSE;   // Positioning request 8: Axis in position
      dbw92 : Int := 2000;   // Time for arm rotation motor stop
      dbw94 : Int := 0;
      dbw96 : Int := 0;
      dbw98 : Int := 0;   // Time for conveyor motor stop
      dbw100 : Int := 0;   // Time for forward on arm rotation and conveyor inverter
      dbw102 : Int := 0;   // Time for backward on arm rotation and conveyor inverter
      dbw104 : Int := 0;
      dbw106 : Int := 0;
      dbw108 : Int := 0;
      dbw110 : Int := 0;
   END_VAR
BEGIN
END_DATA_BLOCK

DATA_BLOCK "DB06_Clamp"   // DB6
{ S7_Optimized_Access := 'FALSE' }
AUTHOR : Robopac
VERSION : 0.0
// stored: AutoNumber false, IsOnlyStoredInLoadMemory false, IsWriteProtectedInAS false
   VAR RETAIN
      dbx0_0 : Bool := FALSE;   // Welder contrast upward
      dbx0_1 : Bool := FALSE;   // Welder contrast downward
      dbx0_2 : Bool := FALSE;   // Welder unit upward
      dbx0_3 : Bool := FALSE;   // Welder unit downward
      dbx0_4 : Bool := FALSE;
      dbx0_5 : Bool := FALSE;   // Film clamp upward
      dbx0_6 : Bool := FALSE;   // Film clamp downward
      dbx0_7 : Bool := FALSE;   // Welder and cut unit forward
      dbx1_0 : Bool := FALSE;   // Welder and cut unit backward
      dbx1_1 : Bool := FALSE;
      dbx1_2 : Bool := FALSE;
      dbx1_3 : Bool := FALSE;
      dbx1_4 : Bool := FALSE;
      dbx1_5 : Bool := FALSE;
      dbx1_6 : Bool := FALSE;
      dbx1_7 : Bool := FALSE;
      dbx2_0 : Bool := FALSE;   // Welder contrast forward
      dbx2_1 : Bool := FALSE;   // Welder contrast backward
      dbx2_2 : Bool := FALSE;
      dbx2_3 : Bool := FALSE;
      dbx2_4 : Bool := FALSE;
      dbx2_5 : Bool := FALSE;
      dbx2_6 : Bool := FALSE;
      dbx2_7 : Bool := FALSE;
      dbb3 : Byte := 16#00;
      dbx4_0 : Bool := FALSE;   // Spool carrage upward to cover tail
      dbx4_1 : Bool := FALSE;   // Spool carrage downward after film tail covered
      dbx4_2 : Bool := FALSE;   // Spool carrage upward at the begining
      dbx4_3 : Bool := FALSE;   // Spool carriage height to pull film at begining
      dbx4_4 : Bool := FALSE;   // Support memory for revolution over welder contrast
      dbx4_5 : Bool := TRUE;   // Clamp carriage is not backward because wrapping cycle
      dbb5 : Byte := 16#00;
      dbw6 : Int := 0;
      dbw8 : Int := 0;
      dbw10 : Int := 500;   // Spool carriage height for film tail airblower
      dbw12 : Int := 0;   // Number of revolution to open clamp
      dbw14 : Int := 0;   // Spool carriage height for film tail wrapped
      dbw16 : Int := 200;   // Spool carriage height to enable revolution over clamp
      dbw18 : Int := 1942;
      dbw20 : Int := 0;
      dbw22 : Int := 0;
      dbw24 : Int := 0;
      dbw26 : Int := 0;
      dbw28 : Int := 0;
      dbw30 : Int := 0;
      dbw32 : Int := 0;
      dbw34 : Int := 0;
      dbw36 : Int := 0;
      dbw38 : Int := 0;
      dbw40 : Int := 0;   // Delay to open clamp (number of 100msec)
      dbw42 : Int := 0;   // Time to open clamp related to actual speed
      dbw44 : Int := 0;
      dbw46 : Int := 0;
      dbw48 : Int := 0;
   END_VAR
BEGIN
END_DATA_BLOCK

DATA_BLOCK "DB07_TopAux"   // DB7
{ S7_Optimized_Access := 'FALSE' }
AUTHOR : Robopac
VERSION : 0.0
// stored: AutoNumber false, IsOnlyStoredInLoadMemory false, IsWriteProtectedInAS false
   VAR RETAIN
      VB700 : Byte := 16#00;
      V701_0 : Bool := TRUE;   // Top film is wrapped
      V701_1 : Bool := FALSE;   // Support memory for top wrapped
      V701_2 : Bool := FALSE;
      V701_3 : Bool := FALSE;
      V701_4 : Bool := FALSE;
      V701_5 : Bool := FALSE;
      V701_6 : Bool := FALSE;
      V701_7 : Bool := FALSE;
   END_VAR
BEGIN
END_DATA_BLOCK

DATA_BLOCK "DB08_Prestretch"   // DB8
{ S7_Optimized_Access := 'FALSE' }
AUTHOR : Robopac
VERSION : 0.0
// stored: AutoNumber false, IsOnlyStoredInLoadMemory false, IsWriteProtectedInAS false
   VAR RETAIN
      dbx0_0 : Bool := FALSE;   // Support memory for prestretch PGSM or PGSA
      dbx0_1 : Bool := FALSE;
      dbx0_2 : Bool := FALSE;
      dbx0_3 : Bool := FALSE;
      dbx0_4 : Bool := FALSE;
      dbx0_5 : Bool := FALSE;
      dbx0_6 : Bool := FALSE;
      dbx0_7 : Bool := FALSE;
      dbw2 : Int := 0;
      dbw4 : Int := 0;
      dbw6 : Int := 0;
      dbw8 : Int := 0;
      dbw10 : Int := 0;   // Film provided for every revolution at max speed (mm per revolution)
      dbw12 : Int := 0;   // Film force value to apply to pallet (mm)
      dbd14 : DInt := 0;   // Support memory for film force to apply to pallet
      dbw18 : Int := 0;   // Film force value to apply to pallet (analog value)
      dbw20 : Int := 0;   // Film force value to apply to pallet (%)
      dbw22 : Int := 0;
      dbw24 : Int := 0;
      dbw26 : Int := 0;
      dbw28 : Int := 0;
      dbw30 : Int := 0;   // Gain for analog scaling
      dbw32 : Int := 200;   // Film prestretch value to apply to pallet
      dbd34 : DInt := 0;   // Support memory for film prestretch to apply to pallet
      dbw38 : Int := 102;   // Film prestretch value to apply to pallet (analog value)
      dbw40 : Int := 0;
      dbw42 : Int := 0;
      dbw44 : Int := 0;
      dbw46 : Int := 0;
      dbw48 : Int := 0;
      dbw50 : Int := 0;   // Support for film prestretch test
      dbw52 : Int := 0;   // Support for film prestretch test
      dbw54 : Int := 0;   // Film weight every mm of film (10^-5 g/mm)
      dbw56 : Int := 0;
      dbw58 : Int := 0;
      dbw60 : Int := 0;
   END_VAR
BEGIN
END_DATA_BLOCK

DATA_BLOCK "DB100_Display"   // DB100
{ S7_Optimized_Access := 'FALSE' }
VERSION : 0.1
// stored: AutoNumber false, IsOnlyStoredInLoadMemory false, IsWriteProtectedInAS false
   VAR RETAIN
      CELLA : Int := 15;   // CELLA (rosa)
      SETPOINT : UInt := 20;   // SETPOINT (rosso)
      PROP : Int := 0;   // PROPORZIONALE (verde)
      "INT" : Int := 0;   // INTEGRALE (giallo)
      FREQ_TIRO : Int := 0;   // U241
      FREQ_PRES : Int := 0;   // U261
   END_VAR
BEGIN
END_DATA_BLOCK

DATA_BLOCK "DB10_ExtConveyors"   // DB10
{ S7_Optimized_Access := 'FALSE' }
VERSION : 0.1
// stored: AutoNumber false, IsOnlyStoredInLoadMemory false, IsWriteProtectedInAS false
   VAR RETAIN
      V1000_0 : Bool := FALSE;
      V1000_1 : Bool := FALSE;
      V1000_2 : Bool := FALSE;
      V1000_3 : Bool := FALSE;
      V1000_4 : Bool := FALSE;
      V1000_5 : Bool := FALSE;
      V1000_6 : Bool := FALSE;
      V1000_7 : Bool := FALSE;
      V1001_0 : Bool := FALSE;
      V1001_1 : Bool := FALSE;
      V1001_2 : Bool := FALSE;
      V1001_3 : Bool := FALSE;
      V1001_4 : Bool := FALSE;
      V1001_5 : Bool := FALSE;
      V1001_6 : Bool := FALSE;
      V1001_7 : Bool := FALSE;
      Out_ConvPos1 : Bool := FALSE;   // Conveyor pos1 motor
      Out_ConvPos2 : Bool := FALSE;   // Conveyor pos2 motor
      Out_ConvPos3 : Bool := FALSE;   // Conveyor pos3 motor
      Out_ConvPos4 : Bool := FALSE;   // Conveyor pos4 motor
      Out_ConvPos5 : Bool := FALSE;   // Conveyor pos5 motor
      Out_ConvPos6 : Bool := FALSE;   // Conveyor pos6 motor
      Out_ConvPos7 : Bool := FALSE;   // Conveyor pos7 motor
      Out_ConvPos8 : Bool := FALSE;   // Conveyor pos8 motor
      Out_ConvPos1Rev : Bool := FALSE;   // Conveyor pos1 motor reverse
      Out_ConvPos2Rev : Bool := FALSE;   // Conveyor pos2 motor reverse
      Out_ConvPos3Rev : Bool := FALSE;   // Conveyor pos3 motor reverse
      Out_ConvPos4Rev : Bool := FALSE;   // Conveyor pos4 motor reverse
      V1003_4 : Bool := FALSE;
      V1003_5 : Bool := FALSE;
      V1003_6 : Bool := FALSE;
      V1003_7 : Bool := FALSE;
      VW1004 : Int := 0;
      Out_ConvPos1X2 : Bool := FALSE;   // Conveyor pos1 motor speed selection X2
      Out_ConvPos2X2 : Bool := FALSE;   // Conveyor pos2 motor speed selection X2
      Out_ConvPos3X2 : Bool := FALSE;   // Conveyor pos3 motor speed selection X2
      Out_ConvPos4X2 : Bool := FALSE;   // Conveyor pos4 motor speed selection X2
      V1006_4 : Bool := FALSE;
      V1006_5 : Bool := FALSE;
      V1006_6 : Bool := FALSE;
      V1006_7 : Bool := FALSE;
      Out_ConvPos2Upw : Bool := FALSE;   // Conveyor pos2 motor upward
      Out_ConvPos2Downw : Bool := FALSE;   // Conveyor pos2 downstroke valve command
      In_ConvPos2Up : Bool := TRUE;   // Conveyor pos2 up photocell NC
      In_ConvPos2Down : Bool := TRUE;   // Conveyor pos2 down photocell NC
      In_ConvPos2ExUp : Bool := TRUE;   // Conveyor pos2 up extrastroke switch NC
      In_ConvPos2Safety : Bool := TRUE;   // Conveyor pos2 down foot safety switch NC
      V1007_6 : Bool := FALSE;
      V1007_7 : Bool := FALSE;
   END_VAR
BEGIN
END_DATA_BLOCK

DATA_BLOCK "DB14_CutWireControl"   // DB14
{ S7_Optimized_Access := 'FALSE' }
VERSION : 0.1
// stored: AutoNumber false, IsOnlyStoredInLoadMemory false, IsWriteProtectedInAS false
   VAR RETAIN
      clean : Time := T#0MS;
      check : Time := T#0MS;
   END_VAR
BEGIN
END_DATA_BLOCK

DATA_BLOCK "DB20_DisplaySysdata"   // DB20
{ S7_Optimized_Access := 'FALSE' }
AUTHOR : Robopac
VERSION : 0.0
// stored: AutoNumber false, IsOnlyStoredInLoadMemory false, IsWriteProtectedInAS false
   VAR RETAIN
      dbd0 : DInt := 238;   // Step for encoder spool carriage movement (mm/100) (Display-Sysadata)
      dbw4 : Int := 6;   // Histeresys for spool carriage positioning (mm) (Display-Sysdata)
      dbw6 : Int := 50;   // Deceleration for spool carriage positioning (mm) (Display-Sysdata)
      dbw8 : Int := 50;   // Low speed for spool carriage movement (%) (Display-Sysdata)
      dbw10 : Int := 100;   // High speed for spool carriage movement (%) (Display-Sysdata)
      dbw12 : Int := 430;   // Spool height (mm) (Display-Sysdata)
      dbw14 : Int := 0;   // Spool carriage down position (mm) (Display-Sysadata)
      dbw16 : Int := 100;   // First step speed for spool carriage movement (%) (Display-Sysadata)
      dbw18 : Int := 240;   // Offset for ftc pallet height (mm) (Display-Sysdata)
      dbw20 : Int := 180;   // Pressure plate height (mm) (Display-Sysdata)
      dbw22 : Int := 7;   // Distance lifter up - conveyor (mm) (Display-Sysdata)
      dbw24 : Int := 0;   // Spool carriage height for film broken cycle (mm) (Display-Sysdata)
      dbw26 : Int := 50;   // Low speed angle to stop rotation (Display-Sysdata)
      dbw28 : Int := 1000;   // Jog1 speed for fast prestretch rool (Display-Sysadata)
      dbw30 : Int := 45;   // Offset for SCSP/2 (Display-Sysadata)
      dbw32 : Int := 78;
      dbw34 : Int := 1100;   // Arm rotation motor and gearbox type (Display-Sysdata)
      dbw36 : Int := 0;   // Delay for test cycle (Display-Sysdata)
      dbx38_0 : Bool := FALSE;   // Film ended or broken cycle included/excluded(1) (Display-Sysdata)
      dbx38_1 : Bool := FALSE;   // Conveyor encoder alarm included(0)/excluded (Display-Sysdata)
      dbx38_2 : Bool := FALSE;   // Test cycle included(1)/excluded (Display-Sysdata)
      dbx38_3 : Bool := FALSE;   // Top film ended or broken included(0)/excluded (Display-Sysdata)
      dbx38_4 : Bool := TRUE;   // Pallet height with pressure plate priority (Display-Sysdata)
      dbx38_5 : Bool := TRUE;   // Spool carriage upward during arm deceleration excluded/included(1) (Display-Sys
      dbx38_6 : Bool := FALSE;   // Pressure plate upward before(0)/after cut cycle (Display-Sysdata)
      dbx38_7 : Bool := FALSE;   // Bit stop pallet infeed (Display-Sysdata)
      dbx39_0 : Bool := FALSE;   // Timeout included/excluded(1) (Display-Sysdata)
      dbx39_1 : Bool := FALSE;   // Reverse cycle request from hmi (Display-Main page)
      dbx39_2 : Bool := FALSE;
      dbx39_3 : Bool := FALSE;
      dbx39_4 : Bool := FALSE;
      dbx39_5 : Bool := FALSE;
      dbx39_6 : Bool := TRUE;   // Top fast cycle
      dbx39_7 : Bool := FALSE;
      dbw40 : Int := 65;   // Spool carriage upward during arm deceleration (mm) (Display-Sysdata)
      dbw42 : Int := 1360;   // Step for infeed conveyor encoder (mm/100) (Display-Sysdata)
      dbw44 : Int := -210;   // Pulse offset for rotation encoder (Display-Sysdata)
      dbw46 : Int := 0;   // Pallet lenght for small pallet (Display-Sysdata)
      dbw48 : Int := 0;   // Decentering for pallet positioning (Display-Sysdata)
      dbw50 : Int := 500;   // Quote for airblower on (mm) (Display-Sysdata)
      dbw52 : Int := 0;   // Spool carriage up to cover film tail (Display-Sysdata)
      dbw54 : Int := 3000;   // Cutting time (Display-Sysdata)
      dbw56 : Int := 1500;   // MAX TIRO SU CELLA (kg) [ex SysdataTempoTwist]
      dbw58 : Int := 2400;   // Delay to open clamp (Display-Sysdata)
      dbw60 : Int := 0;   // Table rotation clampcut phase (°) (Display-Sysdata)
      dbw62 : Int := 200;   // Quote to open clamp (Display-Sysdata)
      dbw64 : Int := 0;   // Step for top carriage forward/backward (mm/100) (Display-Sysdata)
      dbw66 : Int := 1000;   // Step for top carriage upward/downward (mm/100) (Display-Sysdata)
      dbw68 : Int := 600;   // Deceleration for top carriage forward/backward (Display-Sysdata)
      dbw70 : Int := 1500;   // Top carriage up position (Display-Sysdata)
      dbw72 : Int := 0;   // Spool carriage position for top cycle (Display-Sysdata)
      dbw74 : Int := 0;   // Delay for spool carriage downward during top cycle (Display-Sysdata)
      dbw76 : Int := 0;   // Tabke rotation load phase (°) (Display-Sysdata)
      dbw78 : Int := 0;   // Table rotation unload phase (°) (Display-Sysdata)
      dbd80 : DInt := 5627;   // Step for encoder table rotation movement (°/p) (Display-Sysdata)
      dbw84 : Int := 18;   // Histeresys for table rotation positioning (°) (Display-Sysdata)
      dbw86 : Int := 2100;   // Deceleration for table rotation positioning (Hz/sec) (Display-Sysdata)
      dbw88 : Int := 10;   // Low speed for table rotation movement (%) (Display-Sysdata)
      dbw90 : Int := 100;   // High speed for table rotation movement (%) (Display-Sysdata)
      dbw92 : Int := 1800;   // Delay to stop top carriage forward for top film broken
      dbw94 : Int := 1000;   // Delay for top pallet height reading photocell (fast cycle)
      dbw96 : Int := 60;
      dbw98 : Int := 20;
   END_VAR
BEGIN
END_DATA_BLOCK

DATA_BLOCK "DB215_ProgramData"   // DB215
TITLE = Program Data
{ S7_Optimized_Access := 'FALSE' }
VERSION : 0.1
// stored: AutoNumber false, IsOnlyStoredInLoadMemory false, IsWriteProtectedInAS false
   VAR RETAIN
      State_Initialization : UInt := 0;
      State_Setup : UInt := 0;
      InverterFault : Bool := FALSE;   // Inverter Fault (F) - Anomalia
      InverterAlarm : Bool := FALSE;   // Inverter Alarm (A) - Avviso
      Keylock : Bool := FALSE;   // Blocco tasti per utente
      ActiveRecipeMLC : Bool := FALSE;   // Multi-Level Control per la ricetta attiva
      Keylock2 : Bool := FALSE;   // Blocco tasti (StateAuto opp. blocco)
      RecipeModified : Bool := FALSE;
      RecipeSave : Bool := FALSE;
      LoadCellConst : Bool := TRUE;   // valore cella costante
      spare_5 : Bool := FALSE;
      spare_6 : Bool := FALSE;
      spare_7 : Bool := FALSE;
      spare_8 : Bool := FALSE;
      spare_9 : Bool := FALSE;
      spare_10 : Bool := FALSE;
      spare_11 : Bool := FALSE;
      spare_12 : Bool := FALSE;
      Offset_Pulses : Int := 0;   // NOT_USED
      Altimeter_Pulses : Int := 442;
      PhotDelay_Pulses : Int := 40;
      Reinforce_Pulses : Int := 0;
      TopFall_Pulses : Int := 134;
      ManRotStep : UInt := 0;
      RotSpeed : Int := 1770;
      CarSpeedUp : Int := 1396;
      CarSpeedDw : Int := 1396;
      Offset_cella : Int := 240;
      EncCarrDir : Int := -1;   // Direzione petalo carrello (1=av;-1=ind)
      EncCarrMax : Int := 603;   // Max altezza carrello (encoder)
      TiroObiettivo : UInt := 0;   // Tiro obiettivo (da chiamata FC300)
      ContaImpulsi : Int := 0;   // Contatore impulsi 20ms (OB30)
      MLC_HeightPulses : Int := 0;   // MLC_Height_Pulses
      MLC_Rounds : Int := 0;   // MLC_rounds
      LoadCellVal_1 : Int := 227;   // valore cella 1
      LoadCellVal_2 : Int := 227;   // valore cella 2
      PropArmMax : Int := 0;   // Costante proporzionalità corrisp. max freq. braccio
      PropCarrMax : Int := 0;   // Costante proporzionalità corrisp. max freq. carrello
      ValOffsetCella : Int := 10;   // Valore per offset cella durante il reset
      RoundTime : UInt := 4000;
      LastRoundTime : UInt := 2000;
      ReinforceTime : UInt := 0;   // [NOT USED]
      pTiro : Array[0..10] of UInt;
      iTiro : Array[0..10] of UInt;
   END_VAR
BEGIN
   pTiro[0] := 70;
   pTiro[1] := 60;
   pTiro[2] := 50;
   pTiro[3] := 45;
   pTiro[4] := 40;
   pTiro[5] := 35;
   pTiro[6] := 30;
   pTiro[7] := 25;
   pTiro[8..10] := 20;
   iTiro[0] := 70;
   iTiro[1] := 60;
   iTiro[2] := 50;
   iTiro[3] := 45;
   iTiro[4] := 40;
   iTiro[5] := 35;
   iTiro[6] := 30;
   iTiro[7] := 25;
   iTiro[8..10] := 20;
END_DATA_BLOCK

